# B&R Automation Studio project SortingStation
Automation Studio 4.12.7.113 SP; Project implementing the sorting station of the cap processing machine; technology packages: mapp 5.24.3, mappCockpit 5.24.4, mappMotion 5.24.1, mappView 5.24.4

## Configuration SortingStation

CPU 5PPC2100.BY44-000, AutomationRuntime I4.83, Build 4.1.2, Safety 0.0, Vc V4.73.2

### Task classes (Cpu.sw)
```
Cyclic#1 (cycle 2000 us, tolerance 0 us):
  Conveyor <- Source.Conveyor.Conveyor.prg
Cyclic#4:
  Comms <- Infrastructure.Comms.Comms.prg
  Automatic <- Source.Automatic.Automatic.prg
  ManualMode <- Source.Manual.ManualMode.prg
  Homing <- Source.Homing.Homing.prg
  Sorter <- Source.Sorter.Sorter.prg
Cyclic#8:
  Recipe <- Infrastructure.Recipe.Recipe.prg
  AlarmHandl <- Infrastructure.Alarms.AlarmHandling.prg
  HMIHelper <- Infrastructure.HMIHelper.HMIHelper.prg
DataObjects: McAcpSys
NcDataObjects: McDriveLog
Binaries: McAcpDrv, udbdef, McAcpSim, mvLoader, arflatprv, McProfGen, mCoWebSc, TCData, FWRules, arcoal, arsvcreg, iomap, asfw, Role, ashwac, sysconf, arconfig, SortConv, ashwd, User, SortRecipe, SortAlaCor, SortSett, SortAlaHis, Settings, Config
Libraries: CoTrace, AsZip, FileIO, runtime, McBase, MpBase, AsOpcUac, AsOpcUas, McAcpAx, McAxis, McStpAx, MpAxis, MpRecipe, sys_lib, MpFile, standard, MpAlarmX, astime, MpServer, asieccon, asbrstr, asio, asepl, asioacc, asusb, arssl, powerlnk, dataobj, aruser
```

### Hardware
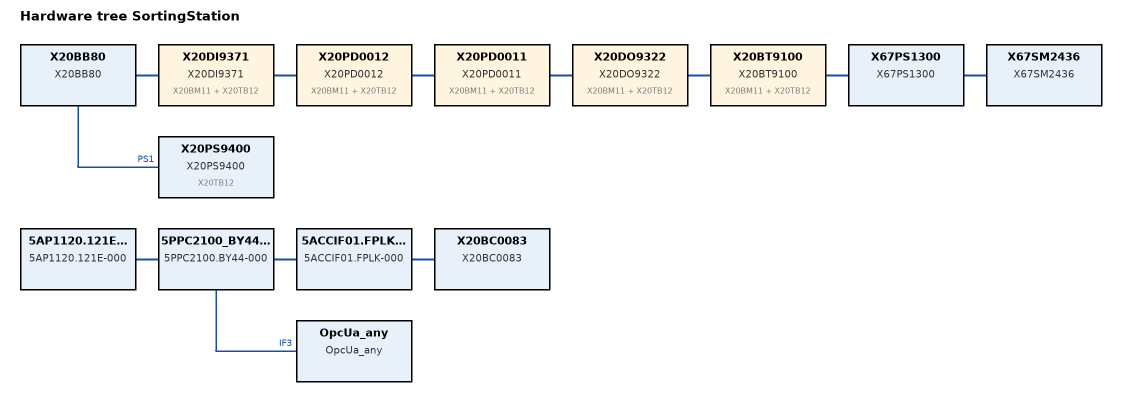
```
5ACCIF01.FPLK-000 : 5ACCIF01.FPLK-000 v1.7.1.0  [SL -> 5PPC2100_BY44_000.SL1]
  Connector IF1:
    ActivateANSL = 1
5AP1120.121E-000 : 5AP1120.121E-000 v2.0.0.0
5PPC2100_BY44_000 : 5PPC2100.BY44-000 v2.1.1.0  [SY -> 5AP1120.121E-000.SY1]
  Connector IF3:
    AssignedOperatingSystem = ARemb
    ActivateDevice = 1
    HostName = sorting-station-ppc2100
    ActivateSnmp = 2
  Connector IF4:
    AssignedOperatingSystem = GPOS
  Connector IF7:
    OperatingSystem = ARemb
    ActivateDevice = 1
    HostName = sorting-station-ppc2100
    Mode = Manual
    InternetAddress = 192.169.0.10
    SubnetMask = 255.255.255.0
    ActivateSnmp = 2
  Connector IF5:
    AssignedOperatingSystem = ARemb
  Connector IF6:
    AssignedOperatingSystem = GPOS
  ConfigurationID = SortingStation_SortingStation
  Cyclic1Duration = 2000
  Cyclic1Tolerance = 0
  FileDevice1
  FileDeviceName1 = USER
  FileDevicePath1 = C:/recipe
  TimeZone = 65
  ActivateDaylightSavingTime = 1
  FtpUser1
  FtpUsername1 = admin  // admin
  FtpUserPassword1 = UdIKPno0znT3css1/ZU0JOxNTb+d8jjj3jhTbXr/0FY=  // admin
  FtpUserSalt1 = m5VJdN1Q
  FTPAccessRight1 = 0
  FTPdevice1 = ALL
  ActivateOpcUa = 1
  OpcUaInformationModels_PV_Version = 1
  ActivateHypervisor = 1
  ARembDramSizeInMb = 512
OpcUa_any : OpcUa_any v1.0.0.1  [ETH1 -> 5PPC2100_BY44_000.IF3 [Cable Type=PowerlinkCable, Length=10, Version=1.0.0.3]]
  ServerDiagnostics = on
  ServerEndpointUrl = opc.tcp://10.67.22.6:4840
  Channel1
  ChannelID1 = ProductAtUnloadingPosition  // Bit from Distribution Station signaling the product is arriving
  ChannelBrowsePath1 = /0:Root/0:Objects/4:PLC/6:Modules/6:&:&:/6:Global PV/6:IO/6:DIn/6:ProductAtUnloadingPosition  // Browse path for the OPCUA node
  Channel2
  ChannelID2 = DistributionReady  // Variable received from Distribution signaling it is ready (no errors)
  ChannelBrowsePath2 = /0:Root/0:Objects/4:PLC/6:Modules/6:&:&:/6:Global PV/6:MachineControl/6:Status/6:ReadyToRun  // Browse path for the OPCUA node
X20BB80 : X20BB80 v1.1.0.0
X20BC0083 : X20BC0083 v2.14.0.0  [PLK1 -> 5ACCIF01.FPLK-000.IF1 (NodeNumber=1) [Cable Type=PowerlinkCable, Length=10, Version=1.0.0.3]; SL -> X20BB80.SL1]
  Supervision = off
X20BM11 : X20BM11 v1.1.0.0  [X2X1 -> X20BB80.IF1]
X20BM11a : X20BM11 v1.1.0.0  [X2X1 -> X20BM11.X2X2]
X20BM11b : X20BM11 v1.1.0.0  [X2X1 -> X20BM11a.X2X2]
X20BM11c : X20BM11 v1.1.0.0  [X2X1 -> X20BM11b.X2X2]
X20BM11d : X20BM11 v1.1.0.0  [X2X1 -> X20BM11c.X2X2]
X20BT9100 : X20BT9100 v1.3.0.0  [SS1 -> X20TB12e.SS; SL -> X20BM11d.SL1]
  Supervision = off
X20DI9371 : X20DI9371 v1.4.0.0  [SS1 -> X20TB12a.SS; SL -> X20BM11.SL1]
  Supervision = off
X20DO9322 : X20DO9322 v1.5.0.0  [SS1 -> X20TB12d.SS; SL -> X20BM11c.SL1]
  Supervision = off
X20PD0011 : X20PD0011 v1.2.0.0  [SS1 -> X20TB12c.SS; SL -> X20BM11b.SL1]
  Supervision = off
X20PD0012 : X20PD0012 v1.2.0.0  [SS1 -> X20TB12b.SS; SL -> X20BM11a.SL1]
  Supervision = off
X20PS9400 : X20PS9400 v1.8.0.0  [SS1 -> X20TB12.SS; PS -> X20BB80.PS1]
  Supervision = off
X20TB12 : X20TB12 v1.0.0.0
X20TB12a : X20TB12 v1.0.0.0
X20TB12b : X20TB12 v1.0.0.0
X20TB12c : X20TB12 v1.0.0.0
X20TB12d : X20TB12 v1.0.0.0
X20TB12e : X20TB12 v1.0.0.0
X67PS1300 : X67PS1300 v1.0.0.0  [X2X1 -> X20BT9100.X2X1 [Cable Type=X2XCable, Length=10, Version=1.0.0.3]]
X67SM2436 : X67SM2436 v2.3.0.0  [X2X1 -> X67PS1300.X2X2 [Cable Type=X2XCable, Length=10, Version=1.0.0.3]]
  Supervision = off
  FunctionModel/DriveConfiguration/Module:
    ActivateModuleSimulationOnPLC = Off
  FunctionModel/DriveConfiguration:
    ModuleParameters = StepperParameters
  FunctionModel/DriveConfiguration/ModuleParameters:
    McStepperTypeID = X67Config
    EncoderType = Incremental
    ReferencePulse = yes
    RatedCurrent = 3.0
    MaximumCurrent = 5.01
    AxesNumber = 2
    FullStepThreshold = 1
    StallDetection = 1
    SmartCurrentControl = 0
    BrakeOutput = 0
    NumberOfDigitalInputs = 6
    NumberOfTriggers = 1
  FunctionModel/DriveConfiguration/Channel[1]/RealAxis:
    AxisReference = gAxisSort
  FunctionModel/DriveConfiguration/Channel[1]/RealAxis/MechanicalElements/Gearbox:
    InputIsReadOnly = 0
    Input = 1
    OutputIsReadOnly = 0
    Output = 1
  FunctionModel/DriveConfiguration/Channel[1]/RealAxis/MechanicalElements/RotaryToLinearTransformation:
    ReferenceDistanceIsReadOnly = 0
    ReferenceDistance = 4
  FunctionModel/DriveConfiguration/Channel[1]/RealAxis/Motor:
    SteppingAngle = 1.8
  FunctionModel/DriveConfiguration/Channel[1]/RealAxis:
    EncoderLink = NoEncoder
  FunctionModel/DriveConfiguration/Channel[1]/RealAxis/Controller:
    ModeIsReadOnly = 0
    Mode = CurrentController
  FunctionModel/DriveConfiguration/Channel[1]/RealAxis/Controller/Mode/Current:
    StandstillCurrent = 1.5
    ConstantSpeedCurrent = 1.5
    SpeedChangeCurrent = 1.5
    FullStepThreshold = 0
    MotorSettlingTime = 1
    DelayedCurrentSwitchOff = 1
  FunctionModel/DriveConfiguration/Channel[1]/RealAxis/Homing:
    Mode = Direct
  FunctionModel/DriveConfiguration/Channel[1]/RealAxis/Homing/Mode:
    Position = 0.0
    ReferencePulse = NotUsed
  FunctionModel/DriveConfiguration/Channel[1]/RealAxis/Homing:
    RestorePositionVariable = 
    ClearPositionError = No
  FunctionModel/DriveConfiguration/Channel[1]/RealAxis/StopReaction:
    DriveError = DecelerationLimit
  FunctionModel/DriveConfiguration/Channel[1]/RealAxis/MovementErrorLimits:
    PositionError = 1.0
    StallDetectionConfiguration = NotUsed
  FunctionModel/DriveConfiguration/Channel[1]/RealAxis:
    JerkFilter = NotUsed
    ZeroVibrationFilter = NotUsed
  FunctionModel/DriveConfiguration/Channel[1]/RealAxis/DigitalInputs/HomingSwitch:
    Source = NotUsed
    Level = High
  FunctionModel/DriveConfiguration/Channel[1]/RealAxis/DigitalInputs/PositiveLimitSwitch:
    Source = NotUsed
    Level = High
  FunctionModel/DriveConfiguration/Channel[1]/RealAxis/DigitalInputs/NegativeLimitSwitch:
    Source = NotUsed
    Level = High
  FunctionModel/DriveConfiguration/Channel[1]/RealAxis/DigitalInputs/Trigger1:
    Source = NotUsed
    Level = High
  FunctionModel/DriveConfiguration/Channel[1]/RealAxis/DigitalInputs/Trigger2:
    Source = NotUsed
    Level = High
  FunctionModel/DriveConfiguration/Channel[1]/RealAxis/DigitalInputs/Quickstop:
    Input = NotUsed
  FunctionModel/DriveConfiguration/Channel[1]/RealAxis/DigitalOutputs:
    BrakeControl = NotUsed
  FunctionModel/DriveConfiguration/Channel[1]/RealAxis/Simulation:
    LoadSimulationMode = NotUsed
  FunctionModel/DriveConfiguration/Channel[2]/RealAxis:
    AxisReference = 
  FunctionModel/DriveConfiguration/Channel[2]/RealAxis/MechanicalElements/Gearbox:
    InputIsReadOnly = 0
    Input = 1
    OutputIsReadOnly = 0
    Output = 1
  FunctionModel/DriveConfiguration/Channel[2]/RealAxis/MechanicalElements/RotaryToLinearTransformation:
    ReferenceDistanceIsReadOnly = 0
    ReferenceDistance = 1
  FunctionModel/DriveConfiguration/Channel[2]/RealAxis/Motor:
    SteppingAngle = 1.8
  FunctionModel/DriveConfiguration/Channel[2]/RealAxis:
    EncoderLink = NoEncoder
  FunctionModel/DriveConfiguration/Channel[2]/RealAxis/Controller:
    ModeIsReadOnly = 0
    Mode = CurrentController
  FunctionModel/DriveConfiguration/Channel[2]/RealAxis/Controller/Mode/Current:
    StandstillCurrent = 0.09
    ConstantSpeedCurrent = 0.45
    SpeedChangeCurrent = 0.9
    FullStepThreshold = 0.0
    MotorSettlingTime = 1
    DelayedCurrentSwitchOff = 1
  FunctionModel/DriveConfiguration/Channel[2]/RealAxis/Homing:
    Mode = Direct
  FunctionModel/DriveConfiguration/Channel[2]/RealAxis/Homing/Mode:
    Position = 0.0
    ReferencePulse = NotUsed
  FunctionModel/DriveConfiguration/Channel[2]/RealAxis/Homing:
    RestorePositionVariable = 
    ClearPositionError = No
  FunctionModel/DriveConfiguration/Channel[2]/RealAxis/StopReaction:
    DriveError = DecelerationLimit
  FunctionModel/DriveConfiguration/Channel[2]/RealAxis/MovementErrorLimits:
    PositionError = 1.0
    StallDetectionConfiguration = NotUsed
  FunctionModel/DriveConfiguration/Channel[2]/RealAxis:
    JerkFilter = NotUsed
    ZeroVibrationFilter = NotUsed
  FunctionModel/DriveConfiguration/Channel[2]/RealAxis/DigitalInputs/HomingSwitch:
    Source = NotUsed
    Level = High
  FunctionModel/DriveConfiguration/Channel[2]/RealAxis/DigitalInputs/PositiveLimitSwitch:
    Source = NotUsed
    Level = High
  FunctionModel/DriveConfiguration/Channel[2]/RealAxis/DigitalInputs/NegativeLimitSwitch:
    Source = NotUsed
    Level = High
  FunctionModel/DriveConfiguration/Channel[2]/RealAxis/DigitalInputs/Trigger1:
    Source = NotUsed
    Level = High
  FunctionModel/DriveConfiguration/Channel[2]/RealAxis/DigitalInputs/Trigger2:
    Source = NotUsed
    Level = High
  FunctionModel/DriveConfiguration/Channel[2]/RealAxis/DigitalInputs/Quickstop:
    Input = NotUsed
  FunctionModel/DriveConfiguration/Channel[2]/RealAxis/DigitalOutputs:
    BrakeControl = NotUsed
  FunctionModel/DriveConfiguration/Channel[2]/RealAxis/Simulation:
    LoadSimulationMode = NotUsed
```

### IoMap.iom - 5PPC2100_BY44_000/IoMap.iom
```iecst
VAR_CONFIG
	::gSorterHardwareIO.DigitalInputs.diProdAvail AT %IX."X20DI9371".DigitalInput01; (*24 VDC, 0.1 to 25 ms switching delay, sink - Product available*)
	::gSorterHardwareIO.DigitalInputs.diMetallic AT %IX."X20DI9371".DigitalInput02; (*24 VDC, 0.1 to 25 ms switching delay, sink - Product is metallic*)
	::gSorterHardwareIO.DigitalInputs.diNotBlack AT %IX."X20DI9371".DigitalInput03; (*24 VDC, 0.1 to 25 ms switching delay, sink - Product is not black*)
	::gSorterHardwareIO.DigitalInputs.diLaneFull AT %IX."X20DI9371".DigitalInput04; (*24 VDC, 0.1 to 25 ms switching delay, sink - Lane full*)
	::gSorterHardwareIO.DigitalInputs.diSwitch1Retracted AT %IX."X20DI9371".DigitalInput05; (*24 VDC, 0.1 to 25 ms switching delay, sink - Switch 1 retracted*)
	::gSorterHardwareIO.DigitalInputs.diSwitch1Extended AT %IX."X20DI9371".DigitalInput06; (*24 VDC, 0.1 to 25 ms switching delay, sink - Switch 1 extended*)
	::gSorterHardwareIO.DigitalInputs.diSwitch2Retracted AT %IX."X20DI9371".DigitalInput07; (*24 VDC, 0.1 to 25 ms switching delay, sink - Switch 2 retracted*)
	::gSorterHardwareIO.DigitalInputs.diSwitch2Extended AT %IX."X20DI9371".DigitalInput08; (*24 VDC, 0.1 to 25 ms switching delay, sink - Switch 2 extended*)
	::gSorterHardwareIO.DigitalOutputs.doExtendSwitch1 AT %QX."X20DO9322".DigitalOutput02; (*24 VDC / 0.5 A, source - Extend switch 1*)
	::gSorterHardwareIO.DigitalOutputs.doExtendSwitch2 AT %QX."X20DO9322".DigitalOutput03; (*24 VDC / 0.5 A, source - Extend switch 2*)
	::gSorterHardwareIO.DigitalOutputs.doRetractStopper AT %QX."X20DO9322".DigitalOutput04; (*24 VDC / 0.5 A, source - Retract stopper*)
	::AlarmHandl:CommsErrors.PLK.FPLK_ModuleOk AT %IX."5ACCIF01.FPLK-000".ModuleOk;
	::AlarmHandl:CommsErrors.X2X.X20BC0083_ModuleOk AT %IX."X20BC0083".ModuleOk;
	::AlarmHandl:CommsErrors.X2X.X20PS9400_ModuleOk AT %IX."X20PS9400".ModuleOk;
	::AlarmHandl:CommsErrors.X2X.X20DI9371_ModuleOk AT %IX."X20DI9371".ModuleOk;
	::AlarmHandl:CommsErrors.X2X.X20PD0012_ModuleOk AT %IX."X20PD0012".ModuleOk;
	::AlarmHandl:CommsErrors.X2X.X20PD0011_ModuleOk AT %IX."X20PD0011".ModuleOk;
	::AlarmHandl:CommsErrors.X2X.X20DO9322_ModuleOk AT %IX."X20DO9322".ModuleOk;
	::AlarmHandl:CommsErrors.X2X.X20BT9100_ModuleOk AT %IX."X20BT9100".ModuleOk;
	::AlarmHandl:CommsErrors.X2X.X67SM2436_ModuleOk AT %IX."X67SM2436".ModuleOk;
	::OpcUaControl.Read.ProductArriving AT %IX."OpcUa_any".ProductAtUnloadingPosition; (*Signal that product is arriving from the distribution station*)
	::OpcUaControl.Read.DistributionReady AT %IX."OpcUa_any".DistributionReady; (*Signal that distribution is without errors and ready to go*)
END_VAR
```

- Physical/SortingStation/5PPC2100_BY44_000/PvMap.vvm: same as Physical/SortingStation/5PPC2100_BY44_000/Cpu.per
### SortConv.axis - 5PPC2100_BY44_000/mappMotion/SortConv.axis
```
Element gAxisSort (Type=axis)
  BaseTypeIsReadOnly = 0
  BaseType = Rotary
    MeasurementUnitIsReadOnly = 0
    MeasurementUnit = 17476
    MeasurementResolutionIsReadOnly = 0
    MeasurementResolution = 0.01
    CountDirectionIsReadOnly = 0
    CountDirection = Standard
  MovementLimitsIsReadOnly = 0
  MovementLimits = Internal
    Position:
      LowerLimitMin = -1.79769313486231E308
      UpperLimitMax = 1.79769313486231E308
      LowerLimit = -1000.0
      UpperLimit = 1000.0
    VelocityIsReadOnly = 0
    Velocity:
      VelocityMax = 3.4E38
      Velocity = 1000
    AccelerationIsReadOnly = 0
    Acceleration:
      AccelerationMax = 3.4E38
      Acceleration = 5000
    DecelerationIsReadOnly = 0
    Deceleration:
      DecelerationMax = 3.4E38
      Deceleration = 5000
  Alarms = None
```

### SortAlaCor.mpalarmxcore - 5PPC2100_BY44_000/mappServices/Alarm/SortAlaCor.mpalarmxcore
```
Element MpLinkSORTING_gAlarmXCore (Type=mpalarmxcore)
  mapp.AlarmX.Core.Configuration:
    [0]:
      Name = Sorting station not homed
      Message = Cannot start automtic mode, the machine needs to be homed first.
      Code = 1001
      Behavior = DiscreteValueMonitoring
        Monitoring:
          MonitoredPV = ::AlarmHandl:CommsErrors.X2X.X20BC0083_ModuleOk
          TriggerValues:
            [0] = FALSE
    [1]:
      Name = Automatic in Error state
      Message = The automatic flow has been stopped, error is present. Please clear error and then re-home machine.
      Code = 1002
    [2]:
      Name = Product stuck between stopper and lane
      Message = The product did not reach the lane, please remove the product and re-home the machine.
      Code = 2001
      Behavior = PersistentAlarm
    [3]:
      Name = Product behind stopper
      Message = Either a second product has come up, or the product did not make it through the stopper after being identified. Please remove the product and rehome the machine.
      Code = 2002
    [4]:
      Name = Incorrect switch open
      Message = If a product is present, you cannot open the correct stopper until the right switch is open. Please see guidelines and try again.
      Code = 3001
    [5]:
      Name = PLK comms error
      Message = There was an error communicating over Powerlink. Please check PLK card and cable connection.
      Code = 4001
    [6]:
      Name = X2X comms error
      Message = There was an error communicating with one of the X20 or X67 modules. Please check connections.
      Code = 4002
    [7]:
      Name = OPCUA comms error
      Message = There was an error in the OPCUA connection. Please check the parameters and re-attempt connection.
```

### SortAlaHis.mpalarmxhistory - 5PPC2100_BY44_000/mappServices/Alarm/SortAlaHis.mpalarmxhistory
```
Element MpLinkSORTING_gAlarmXHistory (Type=mpalarmxhistory)
```

### SortRecipe.mprecipexml - 5PPC2100_BY44_000/mappServices/Recipe/SortRecipe.mprecipexml
```
Element MpLinkSORTING_gRecipeXml (Type=mprecipexml)
```

## Logical view

Binary libraries used (declarations not repeated): operator, runtime, astime, AsIecCon, CoTrace 5.24.4, AsZip, FileIO, McBase 5.24.1, MpBase 5.24.1, AsOpcUac, AsOpcUas, McAcpAx 5.24.1, McAxis 5.24.1, McStpAx 5.24.1, MpAxis 5.24.1, MpRecipe 5.24.3, sys_lib, MpFile 5.24.3, standard, MpAlarmX 5.24.3, MpServer 5.24.0

### Global.typ - Global data types
```iecst
(*global enums*)

TYPE
	gOperatingModeType : 	STRUCT  (*Type for tracking the mode'*)
		AutoMode : BOOL; (*Automatic mode*)
		ManualMode : BOOL; (*Manual mode*)
		HomingMode : BOOL; (*Homing mode*)
	END_STRUCT;
	gOperatingModeEnum :
		( (*Global operating mode*)
		AUTOMATIC := 1, (*Automatic running mode*)
		MANUAL := 2, (*Manual operation mode*)
		HOMING := 3 (*Homing mode*)
		);
END_TYPE

(*global types for sorter hardware*)

TYPE
	gSorterDOType : 	STRUCT  (*Sorter digital output type*)
		doExtendSwitch1 : BOOL; (*Command to extend switch 1*)
		doExtendSwitch2 : BOOL; (*Command to extend switch 2*)
		doRetractStopper : BOOL; (*Retract the stopper*)
	END_STRUCT;
	gSorterDIType : 	STRUCT  (*Sorter digital input type*)
		diProdAvail : BOOL; (*Product available*)
		diMetallic : BOOL; (*Product is metallic*)
		diNotBlack : BOOL; (*Product is not black*)
		diLaneFull : BOOL; (*Lane is full of a product*)
		diSwitch1Retracted : BOOL; (*Switch 1 is retracted*)
		diSwitch1Extended : BOOL; (*Switch 1 is extended*)
		diSwitch2Retracted : BOOL; (*Switch 2 is retracted*)
		diSwitch2Extended : BOOL; (*Switch 2 is extended*)
	END_STRUCT;
	gSorterHardwareIOType : 	STRUCT  (*Hardware IO structure*)
		DigitalOutputs : gSorterDOType; (*Digital outputs*)
		DigitalInputs : gSorterDIType; (*Digital inputs*)
	END_STRUCT;
END_TYPE
```

### Global.var - Global variables
```iecst
(*global variables*)
VAR
	gOperatingMode : gOperatingModeType; (*Mode of operation of the sorting station*)
END_VAR
(*global interface for hardware connect*)
VAR
	gSorterHardwareIO : gSorterHardwareIOType; (*Hardware object for the sorter*)
END_VAR
(*control buttons from main page*)
VAR
	gReset : BOOL; (*Reset/clear button*)
	gStop : BOOL; (*Stop button*)
	gStart : BOOL; (*Start button for the chosen operating mode*)
END_VAR
```


### Package Logical/Source - Package for source code

### Package Logical/Source/Manual - Package for manual mode source code

### ManualIF.typ - Manual interface types
```iecst
(*global interface types*)

TYPE
	ManualCommandType : 	STRUCT  (*Commands type for manual mode*)
		ClassifyProduct : BOOL; (*Command to classify product*)
		JogConveyorBackward : BOOL; (*Jog conveyor forward*)
		JogConveyorForward : BOOL; (*Jog conveyor backward*)
		RetractStopper : BOOL; (*Retract stopper*)
		ExtendSwitch2 : BOOL; (*Extend switch 1*)
		ExtendSwitch1 : BOOL; (*Extend switch 2*)
	END_STRUCT;
	ManualControlType : 	STRUCT  (*Manual mode control structure type*)
		Cmd : ManualCommandType; (*Command for manual mode*)
		Status : ManualStatusType; (*Status for manual mode*)
	END_STRUCT;
	ManualStatusType : 	STRUCT  (*Status type for manual mode*)
		ProductClassified : BOOL; (*Status showing product has been classified*)
		DestinationLane : USINT; (*Lane 1, 2 or 3 - default is 3*)
		ProductInActiveArea : BOOL; (*True if the product is between stopper and lane*)
		Error : BOOL; (*Error triggered*)
	END_STRUCT;
END_TYPE
```

### ManualIF.var - Manual interface variables
```iecst
(*global interface variables*)
VAR
	ManualControl : ManualControlType; (*Control structure for manual mode*)
END_VAR
```

### Program Logical/Source/Manual/ManualMode (IEC) - Manual mode program

#### Cyclic.ld - Cyclic code
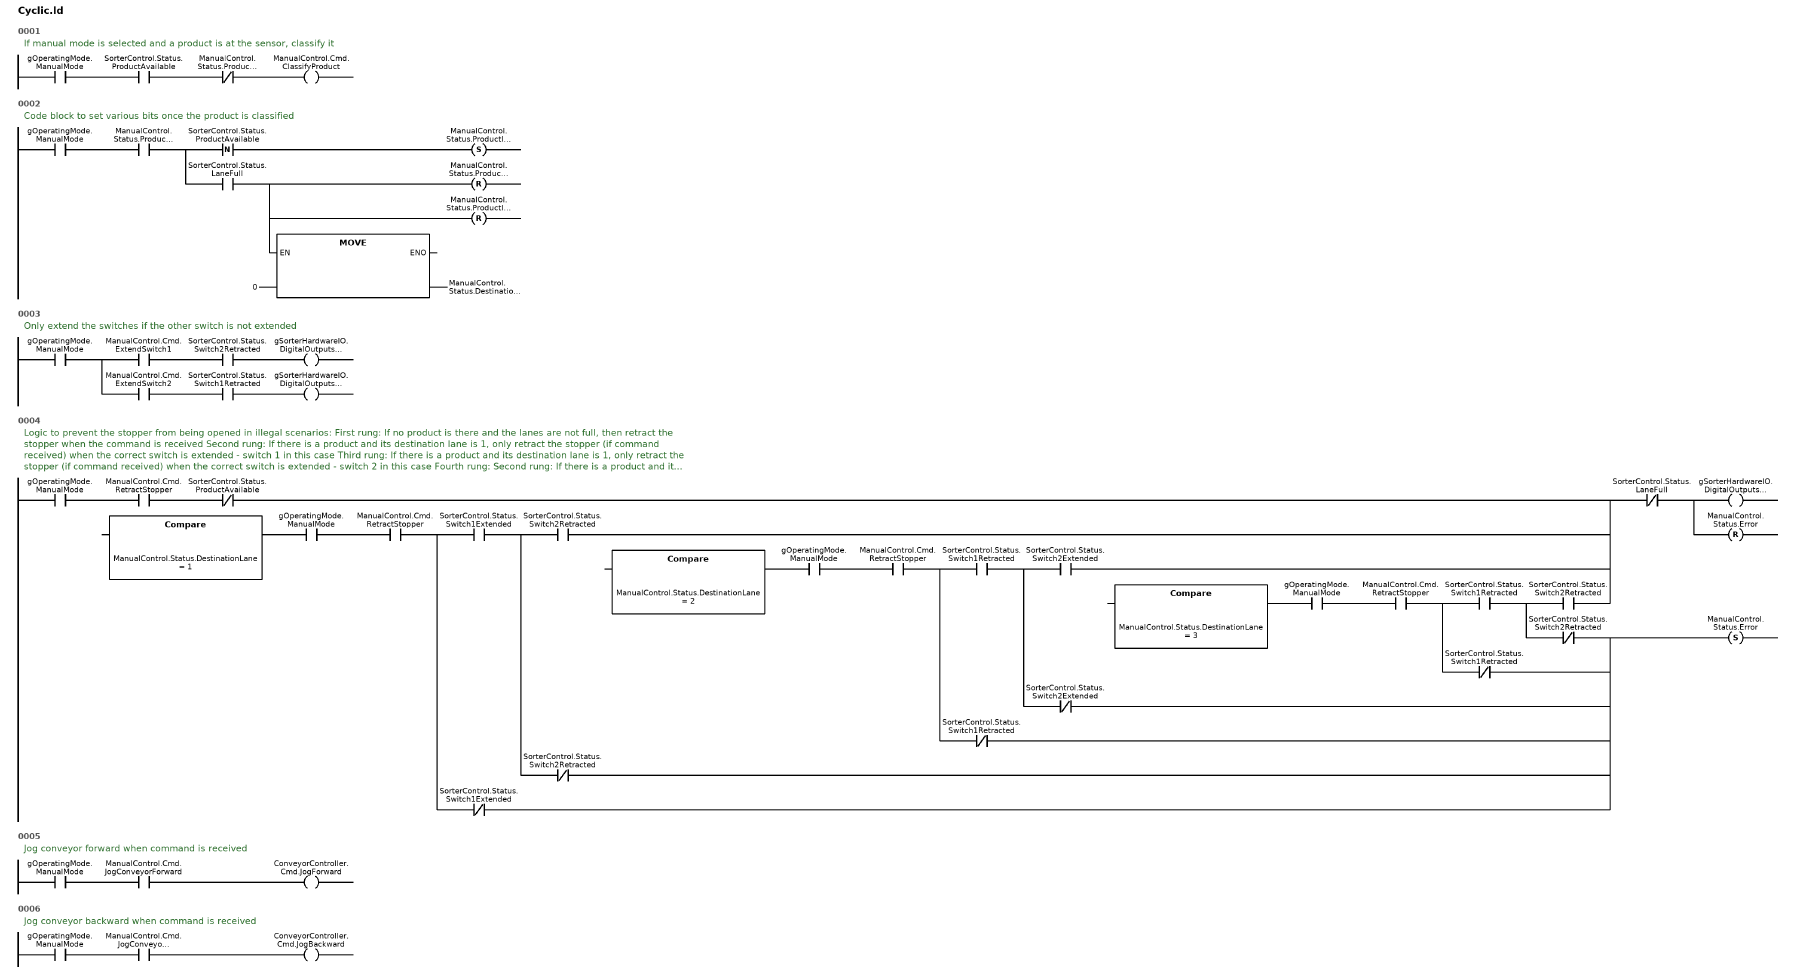
Ladder, written as Structured Text:
```iecst
PROGRAM _CYCLIC
VAR
    _p1 : BOOL;
    _e2 : F_TRIG;
    _p3 : BOOL;
    _p4 : BOOL;
    _p5 : BOOL;
    _p6 : BOOL;
END_VAR
(* Network 1: If manual mode is selected and a product is at the sensor, classify it *)
ManualControl.Cmd.ClassifyProduct := gOperatingMode.ManualMode AND SorterControl.Status.ProductAvailable AND NOT ManualControl.Status.ProductClassified;

(* Network 2: Code block to set various bits once the product is classified *)
_p1 := gOperatingMode.ManualMode AND ManualControl.Status.ProductClassified;
_e2(CLK := SorterControl.Status.ProductAvailable);
IF _p1 AND _e2.Q THEN ManualControl.Status.ProductInActiveArea := TRUE; END_IF;
IF _p1 AND SorterControl.Status.LaneFull THEN
    ManualControl.Status.ProductClassified := FALSE;
    ManualControl.Status.ProductInActiveArea := FALSE;
    ManualControl.Status.DestinationLane := 0;
END_IF;

(* Network 3: Only extend the switches if the other switch is not extended *)
gSorterHardwareIO.DigitalOutputs.doExtendSwitch1 := gOperatingMode.ManualMode AND ManualControl.Cmd.ExtendSwitch1 AND SorterControl.Status.Switch2Retracted;
gSorterHardwareIO.DigitalOutputs.doExtendSwitch2 := gOperatingMode.ManualMode AND ManualControl.Cmd.ExtendSwitch2 AND SorterControl.Status.Switch1Retracted;

(* Network 4: Logic to prevent the stopper from being opened in illegal scenarios: First rung: If no product is there and the lanes are not full, then retract the stopper when the command is received Second rung: If there is a product and its destination lane is 1, only retract the stopper (if command received) when the correct switch is extended - switch 1 in this case Third rung: If there is a product and its destination lane is 1, only retract the stopper (if command received) when the correct switch is extended - switch 2 in this case Fourth rung: Second rung: If there is a product and its destination lane is 1, only retract the stopper (if command received) when no switches are extended Trigger an error in other cases *)
_p3 := (ManualControl.Status.DestinationLane = 1) AND gOperatingMode.ManualMode AND ManualControl.Cmd.RetractStopper;
_p4 := (ManualControl.Status.DestinationLane = 2) AND gOperatingMode.ManualMode AND ManualControl.Cmd.RetractStopper;
_p5 := (ManualControl.Status.DestinationLane = 3) AND gOperatingMode.ManualMode AND ManualControl.Cmd.RetractStopper;
_p6 := ((gOperatingMode.ManualMode AND ManualControl.Cmd.RetractStopper AND NOT SorterControl.Status.ProductAvailable) OR (_p3 AND SorterControl.Status.Switch1Extended AND SorterControl.Status.Switch2Retracted) OR (_p4 AND SorterControl.Status.Switch1Retracted AND SorterControl.Status.Switch2Extended) OR (_p5 AND SorterControl.Status.Switch1Retracted AND SorterControl.Status.Switch2Retracted)) AND NOT SorterControl.Status.LaneFull;
gSorterHardwareIO.DigitalOutputs.doRetractStopper := _p6;
IF _p6 THEN ManualControl.Status.Error := FALSE; END_IF;
IF (_p5 AND ((SorterControl.Status.Switch1Retracted AND NOT SorterControl.Status.Switch2Retracted) OR NOT SorterControl.Status.Switch1Retracted)) OR (_p4 AND ((SorterControl.Status.Switch1Retracted AND NOT SorterControl.Status.Switch2Extended) OR NOT SorterControl.Status.Switch1Retracted)) OR (_p3 AND ((SorterControl.Status.Switch1Extended AND NOT SorterControl.Status.Switch2Retracted) OR NOT SorterControl.Status.Switch1Extended)) THEN
    ManualControl.Status.Error := TRUE;
END_IF;

(* Network 5: Jog conveyor forward when command is received *)
ConveyorController.Cmd.JogForward := gOperatingMode.ManualMode AND ManualControl.Cmd.JogConveyorForward;

(* Network 6: Jog conveyor backward when command is received *)
ConveyorController.Cmd.JogBackward := gOperatingMode.ManualMode AND ManualControl.Cmd.JogConveyorBackward;
END_PROGRAM
```

#### Init.ld - Initialization code
Ladder, written as Structured Text:
```iecst
PROGRAM _INIT
END_PROGRAM
```

#### Exit.ld - Exit code
Ladder, written as Structured Text:
```iecst
PROGRAM _EXIT
END_PROGRAM
```

### Package Logical/Source/Automatic - Package for automatic source code

### AutomaticIF.typ - Automatic interface types
```iecst
(*global interface types*)

TYPE
	AutomaticCommandType : 	STRUCT  (*Command type for automatic*)
		EnableTimer : BOOL; (*Enable the timer*)
	END_STRUCT;
	AutomaticErrorType : 	STRUCT  (*Errors in automatic mode*)
		Error1 : BOOL; (*ERROR 1 - cannot start automatic mode before homing the station*)
	END_STRUCT;
	AutomaticStatusType : 	STRUCT  (*Status type for automatic*)
		Errors : AutomaticErrorType; (*Errors in Auto mode*)
		SortingReady : BOOL; (*Ready bit for comms*)
	END_STRUCT;
	AutomaticControlType : 	STRUCT  (*Control structure for automatic mode*)
		Cmd : AutomaticCommandType; (*Commands for automatic mode*)
		Status : AutomaticStatusType; (*Status for automatic mode*)
	END_STRUCT;
	AutomaticGeneralInfoType : 	STRUCT  (*General info structure for variables that need to be retained*)
		ProductsTotal : UINT; (*Total number of products*)
		AutomaticModeTime : TIME; (*Time that it has been in automatic mode*)
	END_STRUCT;
END_TYPE
```

### AutomaticIF.var - Automatic interface variables
```iecst
(*global interface variables*)
VAR
	AutomaticController : AutomaticControlType; (*Control structure for Automatic*)
	AutomaticGeneralInfo : AutomaticGeneralInfoType; (*General info that is retained*)
END_VAR
```

### Program Logical/Source/Automatic/Automatic (IEC) - Automatic program

#### Cyclic.ld - Cyclic code
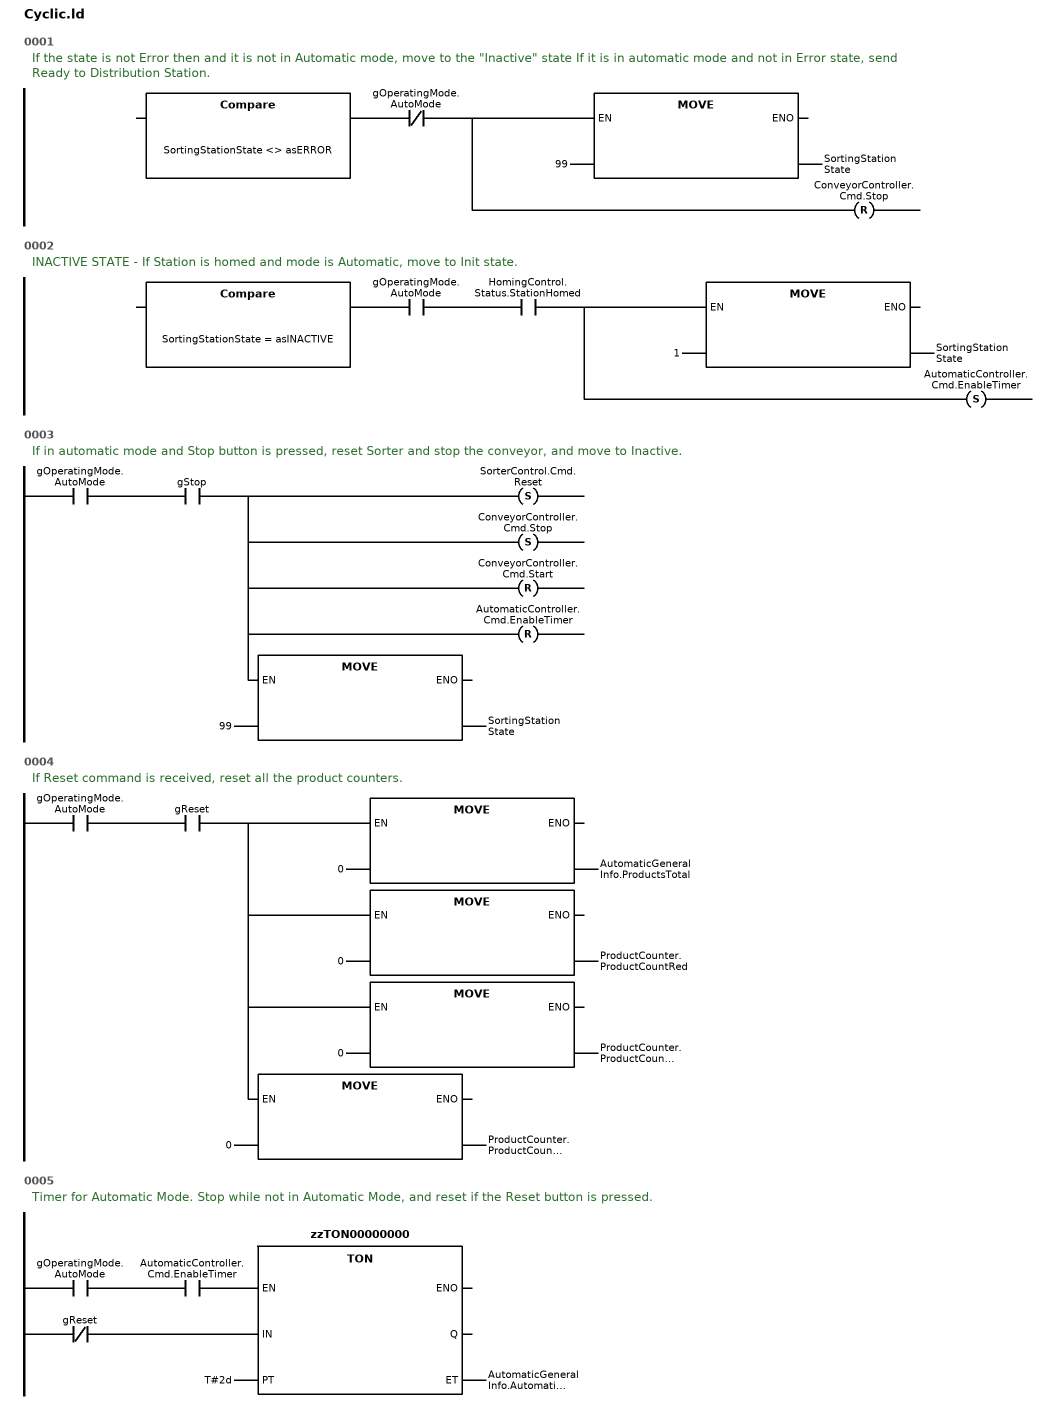
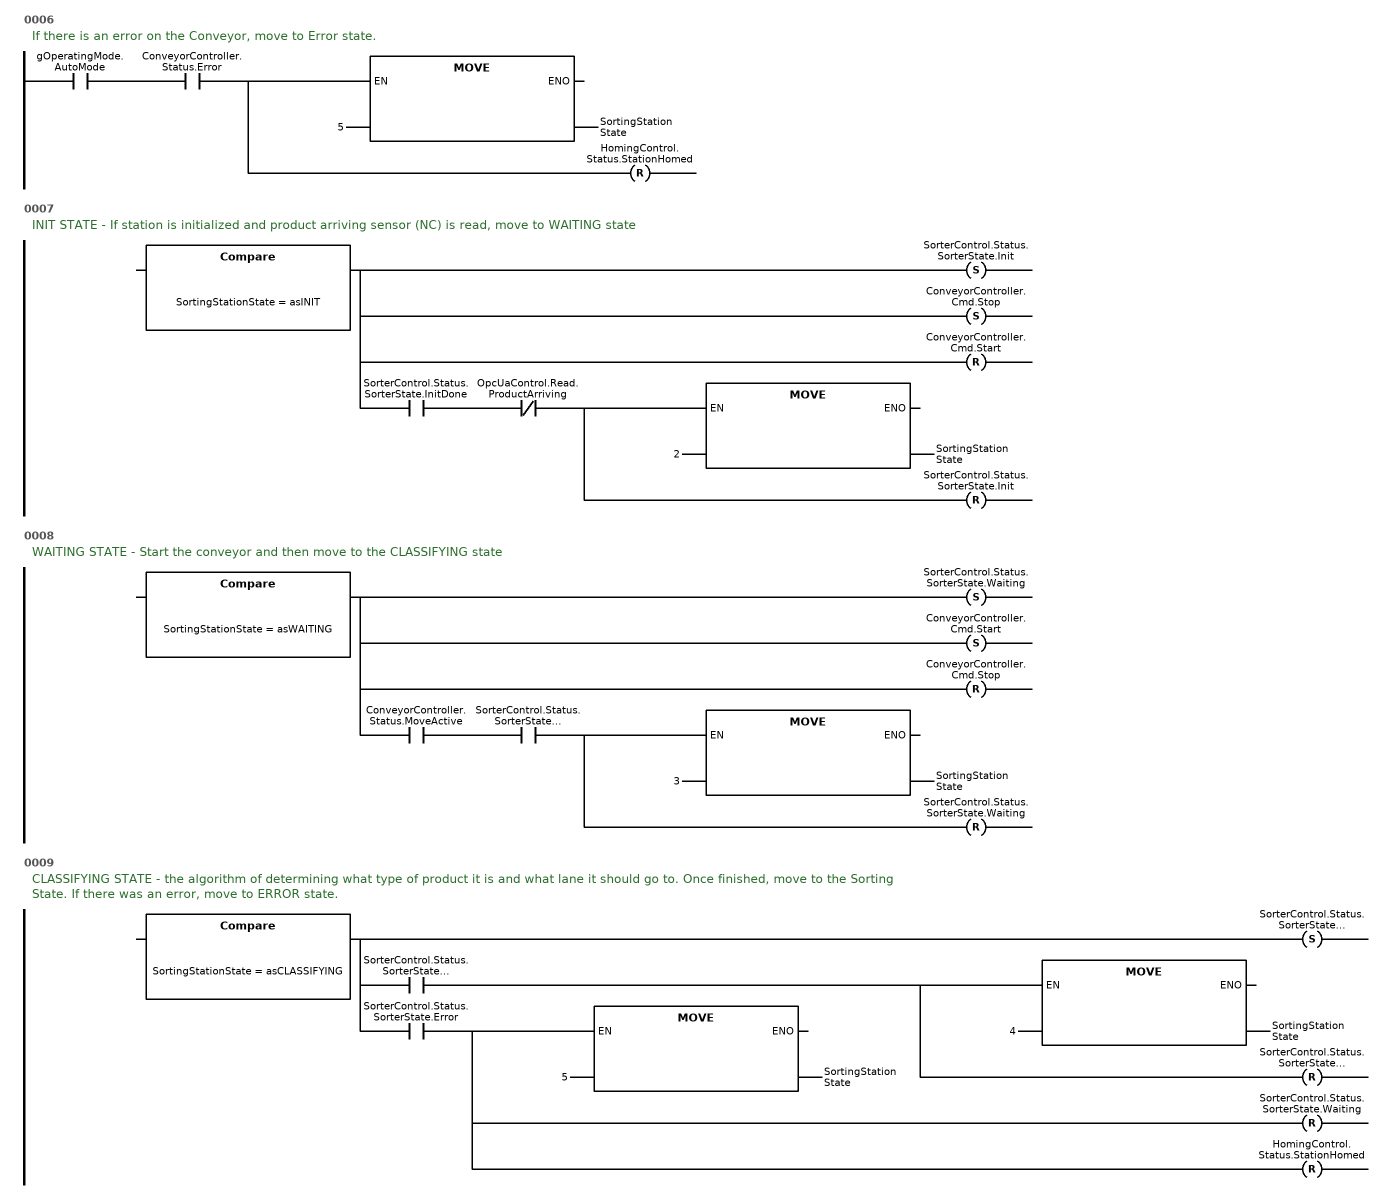
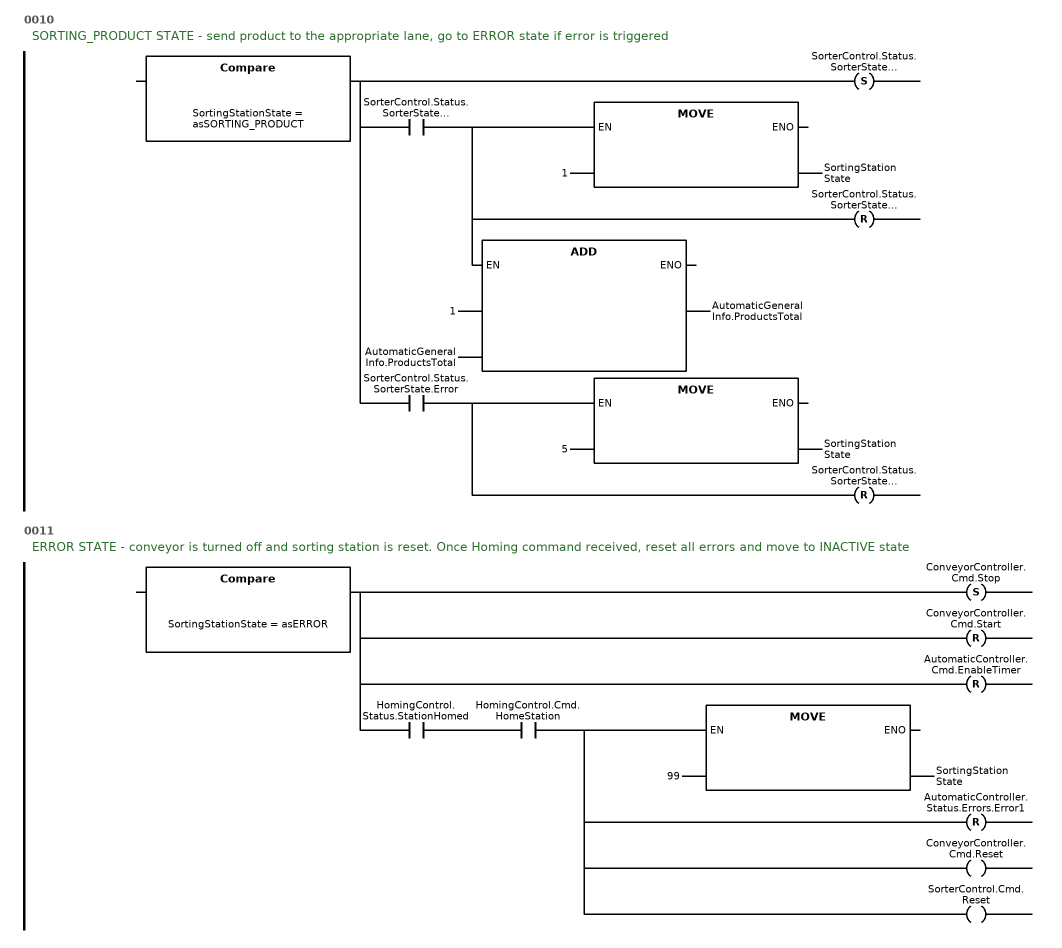
Ladder, written as Structured Text:
```iecst
PROGRAM _CYCLIC
Program to implement state machine for the Automatic Mode
VAR
    _p1 : BOOL;
    _p2 : BOOL;
    _p3 : BOOL;
    _p4 : BOOL;
    _p5 : BOOL;
    _p6 : BOOL;
    _p7 : BOOL;
    _p8 : BOOL;
    _p9 : BOOL;
    _p10 : BOOL;
END_VAR
(* Network 1: If the state is not Error then and it is not in Automatic mode, move to the "Inactive" state If it is in automatic mode and not in Error state, send Ready to Distribution Station. *)
_p1 := (SortingStationState <> asERROR) AND NOT gOperatingMode.AutoMode;
IF _p1 THEN
    SortingStationState := 99;
    ConveyorController.Cmd.Stop := FALSE;
END_IF;

(* Network 2: INACTIVE STATE - If Station is homed and mode is Automatic, move to Init state. *)
_p2 := (SortingStationState = asINACTIVE) AND gOperatingMode.AutoMode AND HomingControl.Status.StationHomed;
IF _p2 THEN
    SortingStationState := 1;
    AutomaticController.Cmd.EnableTimer := TRUE;
END_IF;

(* Network 3: If in automatic mode and Stop button is pressed, reset Sorter and stop the conveyor, and move to Inactive. *)
IF gOperatingMode.AutoMode AND gStop THEN
    SorterControl.Cmd.Reset := TRUE;
    ConveyorController.Cmd.Stop := TRUE;
    ConveyorController.Cmd.Start := FALSE;
    AutomaticController.Cmd.EnableTimer := FALSE;
    SortingStationState := 99;
END_IF;

(* Network 4: If Reset command is received, reset all the product counters. *)
IF gOperatingMode.AutoMode AND gReset THEN
    AutomaticGeneralInfo.ProductsTotal := 0;
    ProductCounter.ProductCountRed := 0;
    ProductCounter.ProductCountBlack := 0;
    ProductCounter.ProductCountMetal := 0;
END_IF;

(* Network 5: Timer for Automatic Mode. Stop while not in Automatic Mode, and reset if the Reset button is pressed. *)
IF gOperatingMode.AutoMode AND AutomaticController.Cmd.EnableTimer THEN
    zzTON00000000(IN := NOT gReset, PT := T#2d);
    AutomaticGeneralInfo.AutomaticModeTime := zzTON00000000.ET;
END_IF;

(* Network 6: If there is an error on the Conveyor, move to Error state. *)
_p3 := gOperatingMode.AutoMode AND ConveyorController.Status.Error;
IF _p3 THEN
    SortingStationState := 5;
    HomingControl.Status.StationHomed := FALSE;
END_IF;

(* Network 7: INIT STATE - If station is initialized and product arriving sensor (NC) is read, move to WAITING state *)
IF (SortingStationState = asINIT) THEN
    SorterControl.Status.SorterState.Init := TRUE;
    ConveyorController.Cmd.Stop := TRUE;
    ConveyorController.Cmd.Start := FALSE;
END_IF;
_p4 := (SortingStationState = asINIT) AND SorterControl.Status.SorterState.InitDone AND NOT OpcUaControl.Read.ProductArriving;
IF _p4 THEN
    SortingStationState := 2;
    SorterControl.Status.SorterState.Init := FALSE;
END_IF;

(* Network 8: WAITING STATE - Start the conveyor and then move to the CLASSIFYING state *)
IF (SortingStationState = asWAITING) THEN
    SorterControl.Status.SorterState.Waiting := TRUE;
    ConveyorController.Cmd.Start := TRUE;
    ConveyorController.Cmd.Stop := FALSE;
END_IF;
_p5 := (SortingStationState = asWAITING) AND ConveyorController.Status.MoveActive AND SorterControl.Status.SorterState.WaitingDone;
IF _p5 THEN
    SortingStationState := 3;
    SorterControl.Status.SorterState.Waiting := FALSE;
END_IF;

(* Network 9: CLASSIFYING STATE - the algorithm of determining what type of product it is and what lane it should go to. Once finished, move to the Sorting State. If there was an error, move to ERROR state. *)
IF (SortingStationState = asCLASSIFYING) THEN
    SorterControl.Status.SorterState.Classifying := TRUE;
END_IF;
_p6 := (SortingStationState = asCLASSIFYING) AND SorterControl.Status.SorterState.ClassifyingDone;
IF _p6 THEN SortingStationState := 4; END_IF;
_p7 := (SortingStationState = asCLASSIFYING) AND SorterControl.Status.SorterState.Error;
IF _p7 THEN SortingStationState := 5; END_IF;
IF _p6 THEN SorterControl.Status.SorterState.Classifying := FALSE; END_IF;
IF _p7 THEN
    SorterControl.Status.SorterState.Waiting := FALSE;
    HomingControl.Status.StationHomed := FALSE;
END_IF;

(* Network 10: SORTING_PRODUCT STATE - send product to the appropriate lane, go to ERROR state if error is triggered *)
IF (SortingStationState = asSORTING_PRODUCT) THEN
    SorterControl.Status.SorterState.SortingProduct := TRUE;
END_IF;
_p8 := (SortingStationState = asSORTING_PRODUCT) AND SorterControl.Status.SorterState.SortingProductDone;
IF _p8 THEN
    SortingStationState := 1;
    SorterControl.Status.SorterState.SortingProduct := FALSE;
    AutomaticGeneralInfo.ProductsTotal := 1 + AutomaticGeneralInfo.ProductsTotal;
END_IF;
_p9 := (SortingStationState = asSORTING_PRODUCT) AND SorterControl.Status.SorterState.Error;
IF _p9 THEN
    SortingStationState := 5;
    SorterControl.Status.SorterState.SortingProduct := FALSE;
END_IF;

(* Network 11: ERROR STATE - conveyor is turned off and sorting station is reset. Once Homing command received, reset all errors and move to INACTIVE state *)
IF (SortingStationState = asERROR) THEN
    ConveyorController.Cmd.Stop := TRUE;
    ConveyorController.Cmd.Start := FALSE;
    AutomaticController.Cmd.EnableTimer := FALSE;
END_IF;
_p10 := (SortingStationState = asERROR) AND HomingControl.Status.StationHomed AND HomingControl.Cmd.HomeStation;
IF _p10 THEN
    SortingStationState := 99;
    AutomaticController.Status.Errors.Error1 := FALSE;
END_IF;
ConveyorController.Cmd.Reset := _p10;
SorterControl.Cmd.Reset := _p10;
END_PROGRAM
```

#### Init.ld - Initialization code
Ladder, written as Structured Text:
```iecst
PROGRAM _INIT
END_PROGRAM
```

#### Exit.ld - Exit code
Ladder, written as Structured Text:
```iecst
PROGRAM _EXIT
END_PROGRAM
```

#### Types.typ - Local data types
```iecst
(*state machine enumerator*)

TYPE
	AutomaticSortingEnum :
		( (*Enum for state machine*)
		asINIT := 1, (*Initial state, homing and setting variables and waiting for start signal*)
		asWAITING := 2, (*Waiting for product to arrive*)
		asCLASSIFYING := 3, (*Identifying and classifying product*)
		asSORTING_PRODUCT := 4, (*Sorting product*)
		asERROR := 5, (*Error state*)
		asINACTIVE := 99
		);
END_TYPE
```

#### Variables.var - Local variables
```iecst
(*local enum*)
VAR
	SortingStationState : AutomaticSortingEnum := asINACTIVE; (*Enumerator to track the state*)
END_VAR
```

### Package Logical/Source/Homing - Package for homing mode

### HomingIF.typ - Homing interface types
```iecst
(*global interface types*)

TYPE
	HomingCommandType : 	STRUCT  (*Commands for homing*)
		HomeStation : BOOL; (*Command to home*)
	END_STRUCT;
	HomingStatusType : 	STRUCT  (*Statuses for homing*)
		StationHomed : BOOL; (*Station is homed*)
	END_STRUCT;
	HomingControlType : 	STRUCT  (*Control structure for homing*)
		Cmd : HomingCommandType; (*Homing commands*)
		Status : HomingStatusType; (*Homing statuses*)
	END_STRUCT;
END_TYPE
```

### HomingIF.var - Homing interface variables
```iecst
(*global interface variables*)
VAR
	HomingControl : HomingControlType; (*Homing controller*)
END_VAR
```

### Program Logical/Source/Homing/Homing (IEC) - Homing task

#### Cyclic.ld - Cyclic code
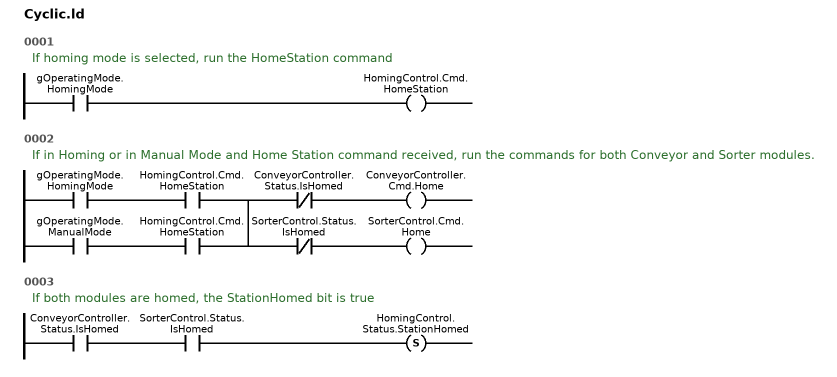
Ladder, written as Structured Text:
```iecst
PROGRAM _CYCLIC
VAR
    _p1 : BOOL;
    _p2 : BOOL;
END_VAR
(* Network 1: If homing mode is selected, run the HomeStation command *)
HomingControl.Cmd.HomeStation := gOperatingMode.HomingMode;

(* Network 2: If in Homing or in Manual Mode and Home Station command received, run the commands for both Conveyor and Sorter modules. *)
_p1 := gOperatingMode.HomingMode AND HomingControl.Cmd.HomeStation;
_p2 := gOperatingMode.ManualMode AND HomingControl.Cmd.HomeStation;
ConveyorController.Cmd.Home := (_p1 OR _p2) AND NOT ConveyorController.Status.IsHomed;
SorterControl.Cmd.Home := (_p1 OR _p2) AND NOT SorterControl.Status.IsHomed;

(* Network 3: If both modules are homed, the StationHomed bit is true *)
IF ConveyorController.Status.IsHomed AND SorterControl.Status.IsHomed THEN
    HomingControl.Status.StationHomed := TRUE;
END_IF;
END_PROGRAM
```

#### Init.ld - Initialization code
Ladder, written as Structured Text:
```iecst
PROGRAM _INIT
END_PROGRAM
```

#### Exit.ld - Exit code
Ladder, written as Structured Text:
```iecst
PROGRAM _EXIT
END_PROGRAM
```

### Package Logical/Source/Conveyor - Package for conveyor source code

### ConveyorIF.typ - Conveyor interface types
```iecst
(*global interface structure types*)

TYPE
	ConveyorCommandType : 	STRUCT  (*Conveyor command structure type*)
		Start : BOOL; (*Command to start the conveyor moving*)
		Stop : BOOL; (*Command to stop the conveyor*)
		Reset : BOOL; (*Command to reset in case of an error*)
		JogForward : BOOL; (*Jog command forward*)
		JogBackward : BOOL; (*Jog command backward*)
		Power : BOOL; (*Command to power on the axis*)
		Home : BOOL; (*Command to home the axis*)
	END_STRUCT;
	ConveyorParameterType : 	STRUCT  (*Conveyor parameter structure type*)
		Position : LREAL := 0.0; (*Initial parameter for the axis - position*)
		Velocity : REAL := 400; (*Initial parameter for the axis - velocity*)
		Acceleration : REAL := 3000; (*Initial parameter for the axis - acceleration*)
		Deceleration : REAL := 3000; (*Initial parameter for the axis - deceleration*)
		HomingMode : McHomingModeEnum := mcHOMING_DEFAULT; (*Homing mode*)
	END_STRUCT;
	ConveyorType : 	STRUCT  (*Conveyor controller type*)
		Cmd : ConveyorCommandType; (*Instance of command structure*)
		Par : ConveyorParameterType; (*Instance of parameter structure*)
		Status : ConveyorStatusType; (*Instance of status structure*)
	END_STRUCT;
	ConveyorStatusType : 	STRUCT  (*Conveyor status structure type*)
		IsPowered : BOOL; (*True if powered*)
		IsHomed : BOOL; (*Status variable true if it is homed*)
		Error : BOOL; (*True if there is an error present*)
		MoveActive : BOOL; (*Checking if move is active*)
	END_STRUCT;
END_TYPE
```

### ConveyorIF.var - Conveyor interface varaibles
```iecst
(*global interface variables*)
VAR
	ConveyorController : ConveyorType; (*Conveyor control structure*)
END_VAR
```

### Program Logical/Source/Conveyor/Conveyor (IEC) - Sorting conveyor

#### Cyclic.ld - Cyclic code
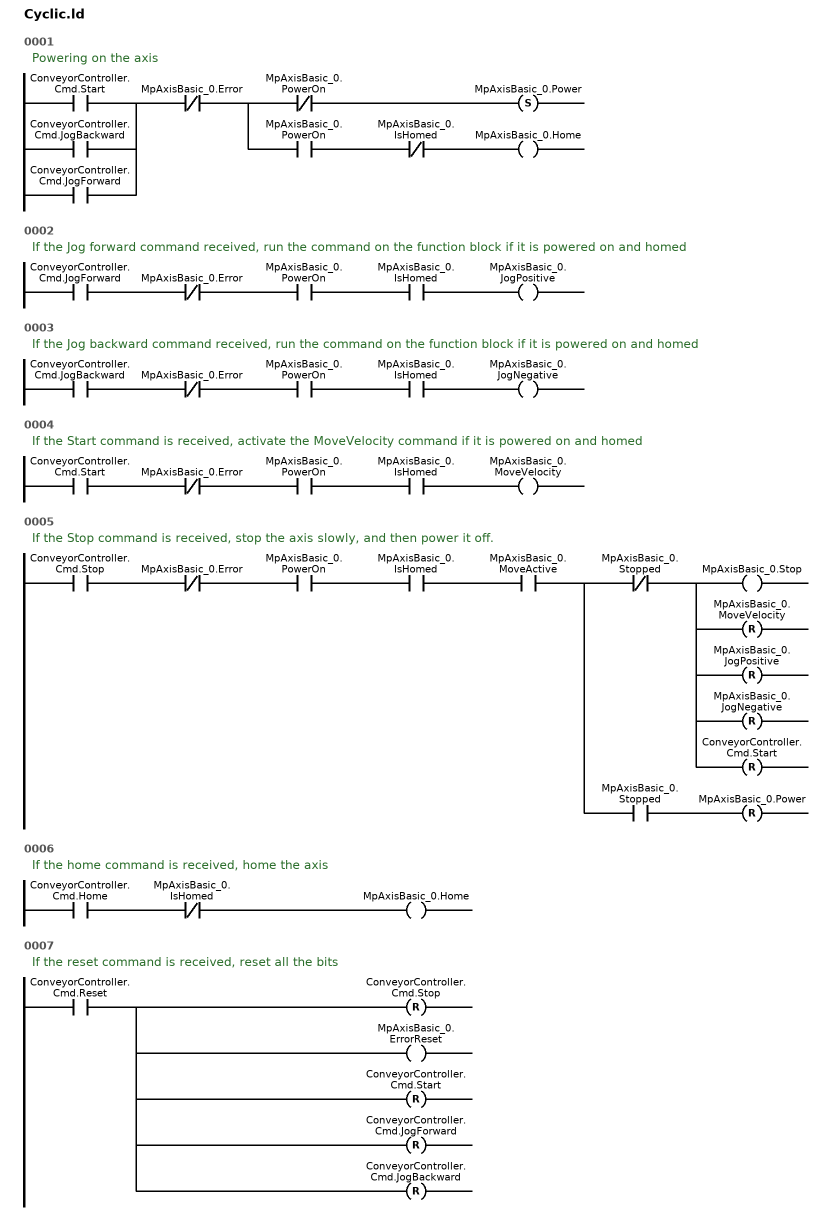
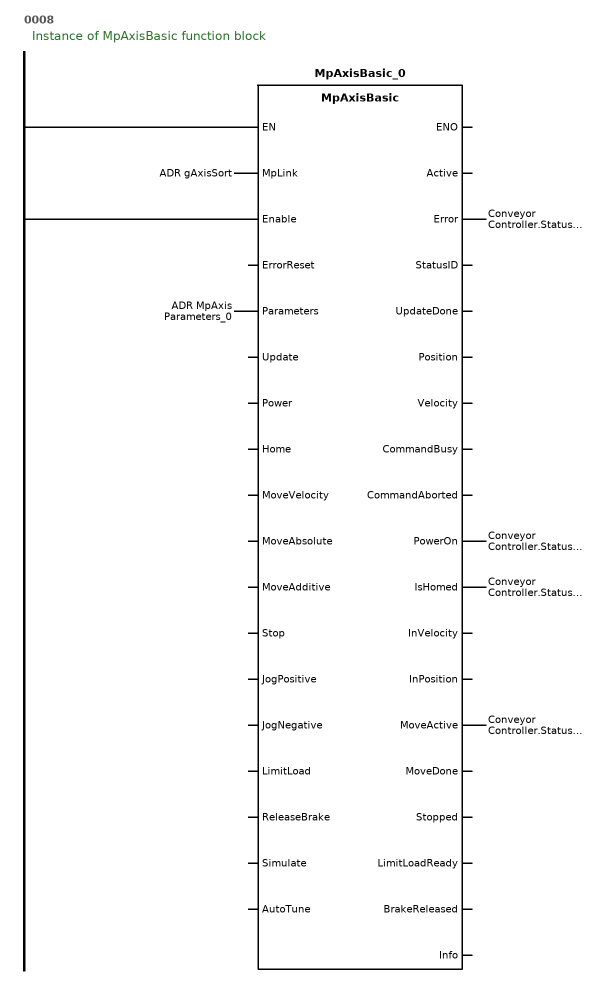
Ladder, written as Structured Text:
```iecst
PROGRAM _CYCLIC
VAR
    _p1 : BOOL;
    _p2 : BOOL;
    _p3 : BOOL;
    _p4 : BOOL;
END_VAR
(* Network 1: Powering on the axis *)
_p1 := (ConveyorController.Cmd.Start OR ConveyorController.Cmd.JogBackward OR ConveyorController.Cmd.JogForward) AND NOT MpAxisBasic_0.Error;
IF _p1 AND NOT MpAxisBasic_0.PowerOn THEN MpAxisBasic_0.Power := TRUE; END_IF;
MpAxisBasic_0.Home := _p1 AND MpAxisBasic_0.PowerOn AND NOT MpAxisBasic_0.IsHomed;

(* Network 2: If the Jog forward command received, run the command on the function block if it is powered on and homed *)
MpAxisBasic_0.JogPositive := ConveyorController.Cmd.JogForward AND NOT MpAxisBasic_0.Error AND MpAxisBasic_0.PowerOn AND MpAxisBasic_0.IsHomed;

(* Network 3: If the Jog backward command received, run the command on the function block if it is powered on and homed *)
MpAxisBasic_0.JogNegative := ConveyorController.Cmd.JogBackward AND NOT MpAxisBasic_0.Error AND MpAxisBasic_0.PowerOn AND MpAxisBasic_0.IsHomed;

(* Network 4: If the Start command is received, activate the MoveVelocity command if it is powered on and homed *)
MpAxisBasic_0.MoveVelocity := ConveyorController.Cmd.Start AND NOT MpAxisBasic_0.Error AND MpAxisBasic_0.PowerOn AND MpAxisBasic_0.IsHomed;

(* Network 5: If the Stop command is received, stop the axis slowly, and then power it off. *)
_p2 := ConveyorController.Cmd.Stop AND NOT MpAxisBasic_0.Error AND MpAxisBasic_0.PowerOn AND MpAxisBasic_0.IsHomed AND MpAxisBasic_0.MoveActive;
_p3 := _p2 AND NOT MpAxisBasic_0.Stopped;
MpAxisBasic_0.Stop := _p2 AND NOT MpAxisBasic_0.Stopped;
IF _p3 THEN
    MpAxisBasic_0.MoveVelocity := FALSE;
    MpAxisBasic_0.JogPositive := FALSE;
    MpAxisBasic_0.JogNegative := FALSE;
    ConveyorController.Cmd.Start := FALSE;
END_IF;
IF _p2 AND MpAxisBasic_0.Stopped THEN MpAxisBasic_0.Power := FALSE; END_IF;

(* Network 6: If the home command is received, home the axis *)
MpAxisBasic_0.Home := ConveyorController.Cmd.Home AND NOT MpAxisBasic_0.IsHomed;

(* Network 7: If the reset command is received, reset all the bits *)
_p4 := ConveyorController.Cmd.Reset;
IF ConveyorController.Cmd.Reset THEN ConveyorController.Cmd.Stop := FALSE; END_IF;
MpAxisBasic_0.ErrorReset := _p4;
IF _p4 THEN
    ConveyorController.Cmd.Start := FALSE;
    ConveyorController.Cmd.JogForward := FALSE;
    ConveyorController.Cmd.JogBackward := FALSE;
END_IF;

(* Network 8: Instance of MpAxisBasic function block *)
MpAxisBasic_0(MpLink := ADR(gAxisSort), Enable := TRUE, Parameters := ADR(MpAxisParameters_0));
ConveyorController.Status.Error := MpAxisBasic_0.Error;
ConveyorController.Status.IsPowered := MpAxisBasic_0.PowerOn;
ConveyorController.Status.IsHomed := MpAxisBasic_0.IsHomed;
ConveyorController.Status.MoveActive := MpAxisBasic_0.MoveActive;
END_PROGRAM
```

#### Init.ld - Initialization code
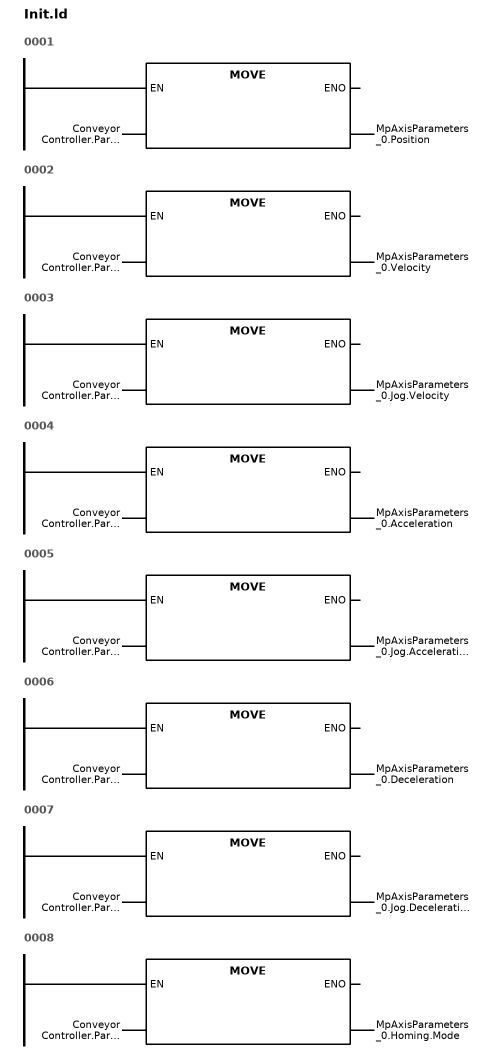
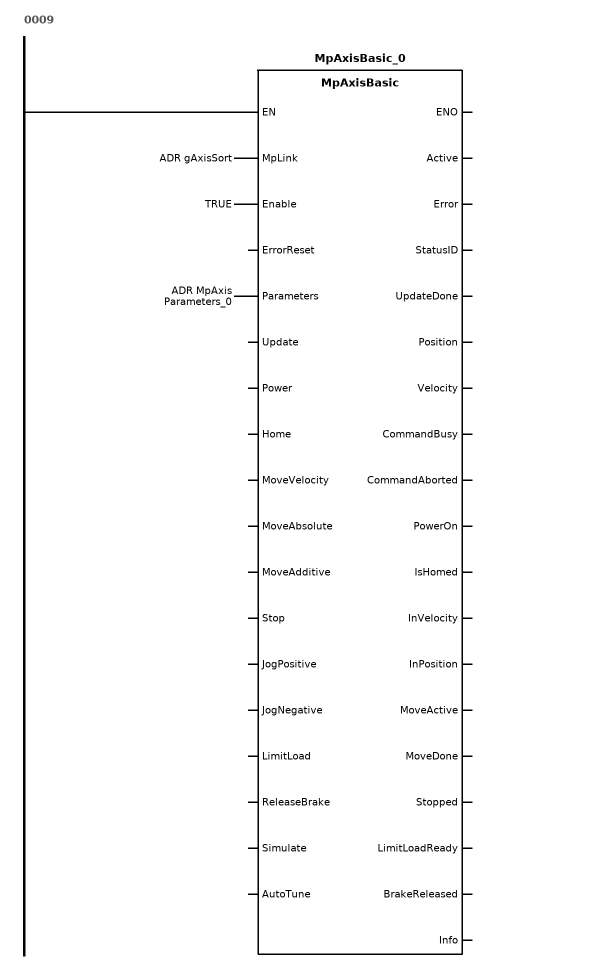
Ladder, written as Structured Text:
```iecst
PROGRAM _INIT
(* Network 1 *)
MpAxisParameters_0.Position := ConveyorController.Par.Position;

(* Network 2 *)
MpAxisParameters_0.Velocity := ConveyorController.Par.Velocity;

(* Network 3 *)
MpAxisParameters_0.Jog.Velocity := ConveyorController.Par.Velocity;

(* Network 4 *)
MpAxisParameters_0.Acceleration := ConveyorController.Par.Acceleration;

(* Network 5 *)
MpAxisParameters_0.Jog.Acceleration := ConveyorController.Par.Acceleration;

(* Network 6 *)
MpAxisParameters_0.Deceleration := ConveyorController.Par.Deceleration;

(* Network 7 *)
MpAxisParameters_0.Jog.Deceleration := ConveyorController.Par.Deceleration;

(* Network 8 *)
MpAxisParameters_0.Homing.Mode := ConveyorController.Par.HomingMode;

(* Network 9 *)
MpAxisBasic_0(MpLink := ADR(gAxisSort), Enable := TRUE, Parameters := ADR(MpAxisParameters_0));
END_PROGRAM
```

#### Exit.ld - Exit code
Ladder, written as Structured Text:
```iecst
PROGRAM _EXIT
END_PROGRAM
```

#### Types.typ - Local data types
```iecst
(*local enumerated types*)

TYPE
	MotionControlEnum :
		( (*Enum type for state machine variable*)
		mcINIT := 1, (*Intial state*)
		mcPOWER := 2, (*Powering on*)
		mcHOME := 3, (*Homing the axis*)
		mcWAIT_FOR_CMD := 4, (*Waiting for a move command*)
		mcPROCESS := 6, (*Process the move command*)
		mcERROR := 7 (*Error handling*)
		);
END_TYPE
```

#### Variables.var - Local variables
```iecst
(*local function blocks*)
VAR
	MpAxisBasic_0 : MpAxisBasic; (*MpAxisBasic function block to control stepper motor*)
END_VAR
(*local structures*)
VAR
	MpAxisParameters_0 : MpAxisBasicParType; (*Parameter structure for the axis*)
END_VAR
(*local enumerators*)
VAR
	MotionControlState : MotionControlEnum := mcINIT; (*Enumerator to keep track of state machine status*)
END_VAR
```

### Package Logical/Source/Sorter - Package for sorter source code

### SorterIF.typ - Interface types for Sorter
```iecst
(*global sorter interface types*)

TYPE
	SorterCommandType : 	STRUCT  (*Commands to pass to the sorter*)
		ExtendSwitch1 : BOOL; (*Command to extend the first switch*)
		ExtendSwitch2 : BOOL; (*Command to extend the second switch*)
		RetractStopper : BOOL; (*Command to retract the stopper*)
		InternalHome : BOOL; (*Separate command to home internally*)
		Home : BOOL; (*Command to home sorter*)
		Reset : BOOL; (*Command to reset*)
	END_STRUCT;
	SortingRecipeType : 	STRUCT  (*Recipe type for lane allocation*)
		Lane1ProductType : ProductTypeEnum; (*Lane 1 product type allocation*)
		Lane2ProductType : ProductTypeEnum; (*Lane 2 product type allocation*)
		Lane3ProductType : ProductTypeEnum; (*Lane 3 product type allocation*)
	END_STRUCT;
	SorterParameterType : 	STRUCT  (*Parameters for the sorter*)
		LaneAllocationRecipe : SortingRecipeType; (*Lane allocation recipe*)
	END_STRUCT;
	SorterErrors : 	STRUCT  (*Structure for the process errors of the sorter*)
		Error1 : BOOL; (*ERROR 1 = Cap not sorted, stuck on conveyor or ejected. Please check machine*)
		Error2 : BOOL; (*ERROR 2 = Cap stuck behind stopped*)
		Error3 : BOOL; (*ERROR 3 = One of the lanes is full*)
	END_STRUCT;
	SorterStates : 	STRUCT  (*Local state machine tracker*)
		Init : BOOL; (*Initial state*)
		InitDone : BOOL; (*Initial done bit*)
		Waiting : BOOL; (*Waiting state*)
		WaitingDone : BOOL; (*Waiting done bit*)
		Classifying : BOOL; (*Classifying state*)
		ClassifyingDone : BOOL; (*Classifying done bit*)
		SortingProduct : BOOL; (*Sorting state*)
		SortingProductDone : BOOL; (*Sorting done bit*)
		Error : BOOL; (*Error state*)
	END_STRUCT;
	SorterStatusType : 	STRUCT  (*Status variables from the sorter*)
		ProductAvailable : BOOL; (*Product is available at beginning of line*)
		ProductMetallic : BOOL; (*Product material sensor*)
		ProductNotBlack : BOOL; (*Product color sensor*)
		ProductType : ProductTypeEnum := ptUNKNOWN; (*Product type*)
		LaneFull : BOOL; (*Product in between stopper and sorting*)
		Switch1Retracted : BOOL; (*Switch 1 is retracted (not active)*)
		Switch1Extended : BOOL; (*Switch 1 is extended (active)*)
		Switch2Retracted : BOOL; (*Switch 2 is retracted (not active)*)
		Switch2Extended : BOOL; (*Switch 2 is extended (active)*)
		IsHomed : BOOL; (*True if all pneumatic valves in home position*)
		ProcessDone : BOOL; (*Process done bit*)
		SorterState : SorterStates; (*State machine local*)
		Errors : SorterErrors; (*Errors structure*)
		DestLane : UINT := 0; (*Destination lane, 1 2 or 3*)
	END_STRUCT;
	SorterType : 	STRUCT  (*Sorter custom type for interface*)
		Cmd : SorterCommandType; (*Command structure for sorter*)
		Par : SorterParameterType; (*Parameter structure for sorter*)
		Status : SorterStatusType; (*Status structure with feedback from sorter*)
	END_STRUCT;
	ProductCounterType : 	STRUCT  (*Product counter type*)
		ProductCountRed : UINT; (*Product counter for red products*)
		ProductCountBlack : UINT; (*Product counter for black products*)
		ProductCountMetal : UINT; (*Product counter for metal products*)
	END_STRUCT;
END_TYPE

(*global sorter enums*)

TYPE
	ProductTypeEnum :
		( (*Enumerator to track type of product*)
		ptUNKNOWN := 1, (*Initial state*)
		ptRED := 2, (*Product is red color and plastic*)
		ptBLACK := 3, (*Product is black color and plastic*)
		ptMETAL := 4 (*Product is metallic*)
		);
END_TYPE
```

### SorterIF.var - Interface variables for Sorter
```iecst
(*global sorter interface variables*)
VAR
	SorterControl : SorterType; (*Control structure for the Sorter*)
	ProductCounter : ProductCounterType; (*Counters for all three product types*)
END_VAR
```

### Program Logical/Source/Sorter/Sorter (IEC) - Sorter program

#### Cyclic.ld - Cyclic code
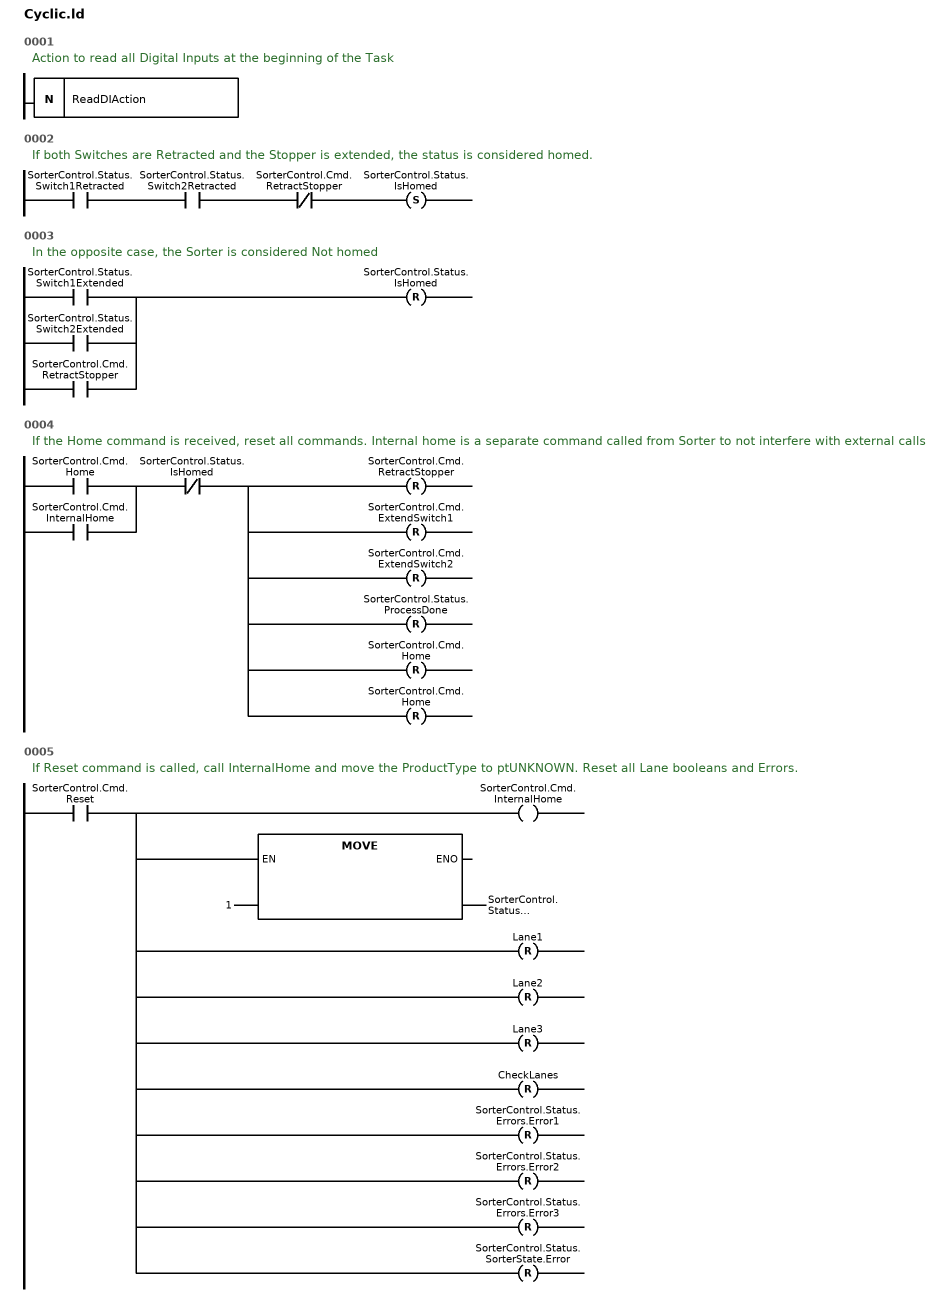
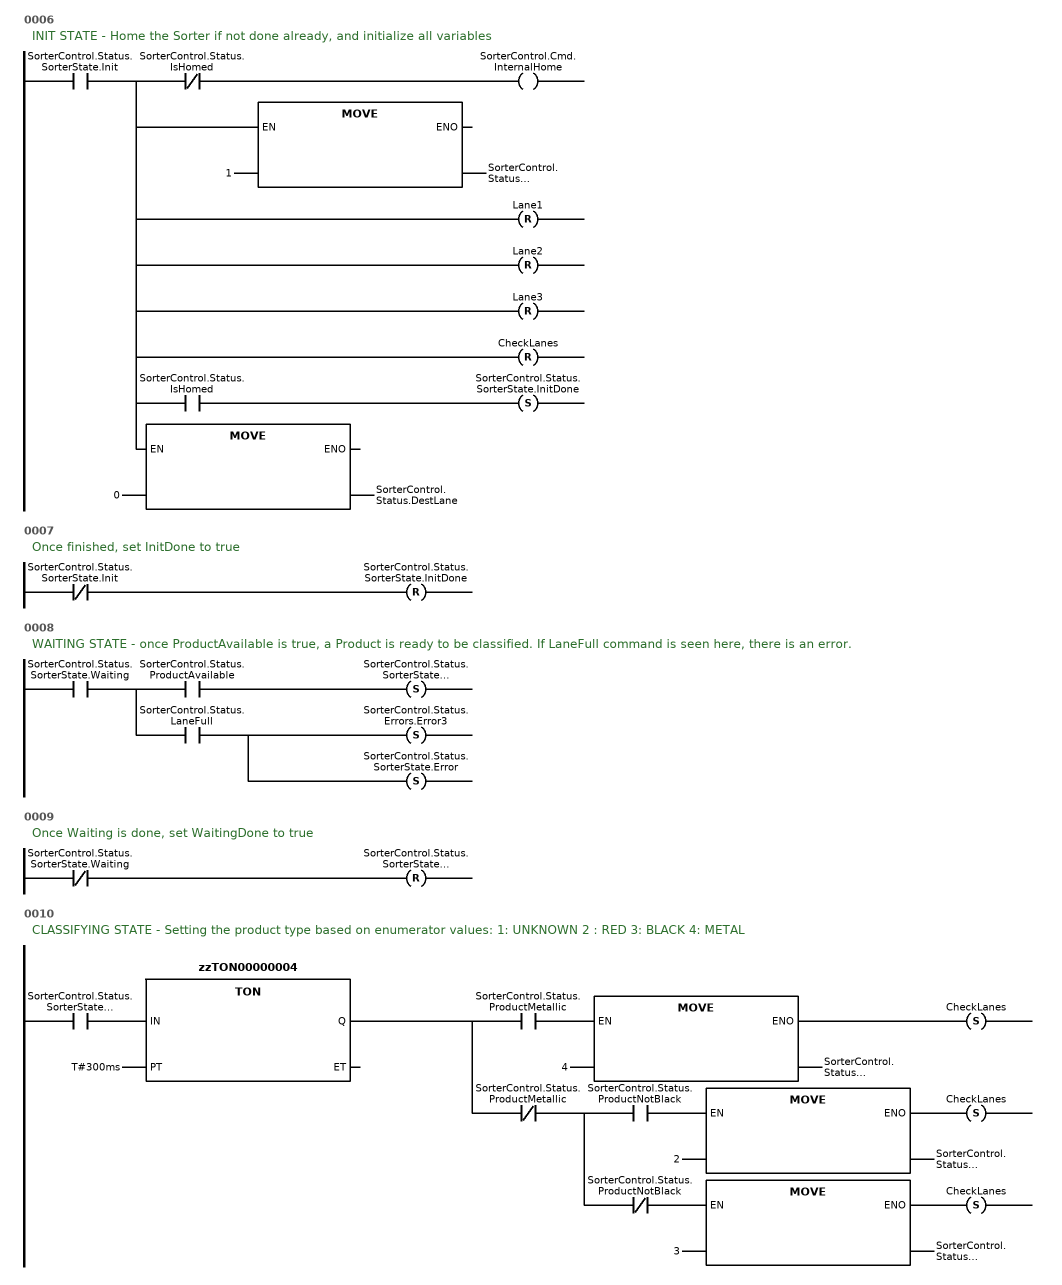
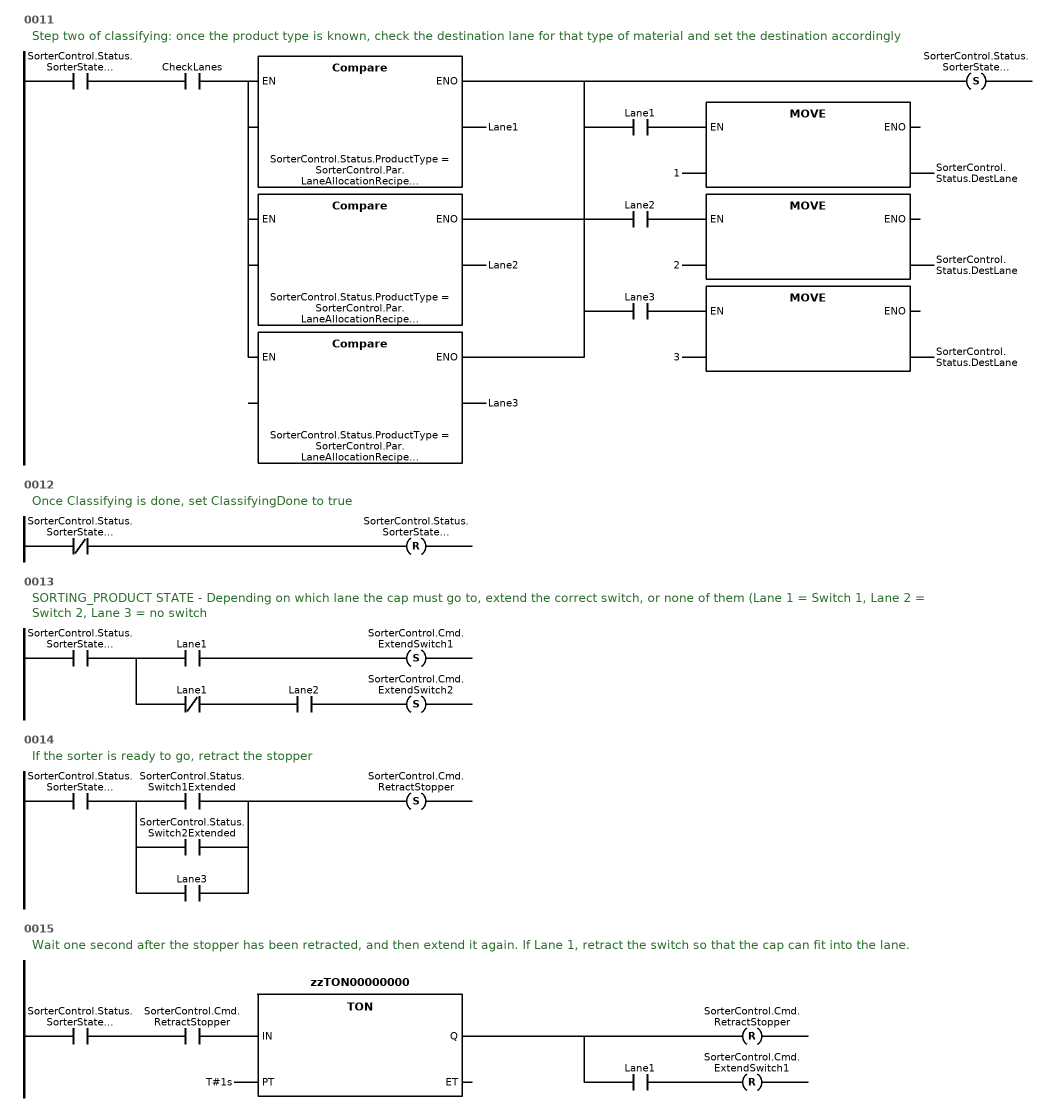
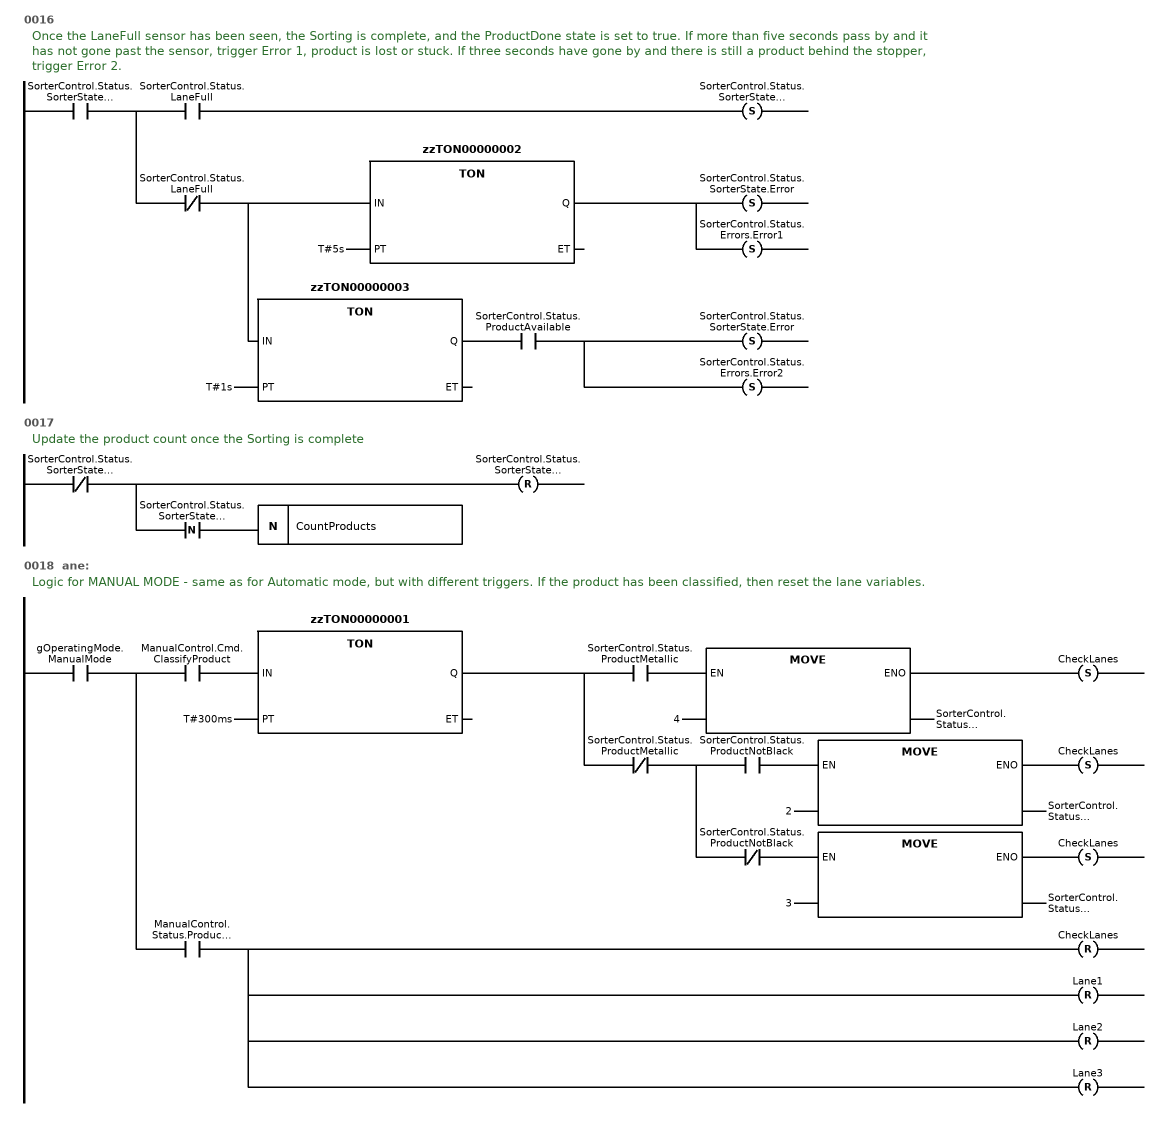
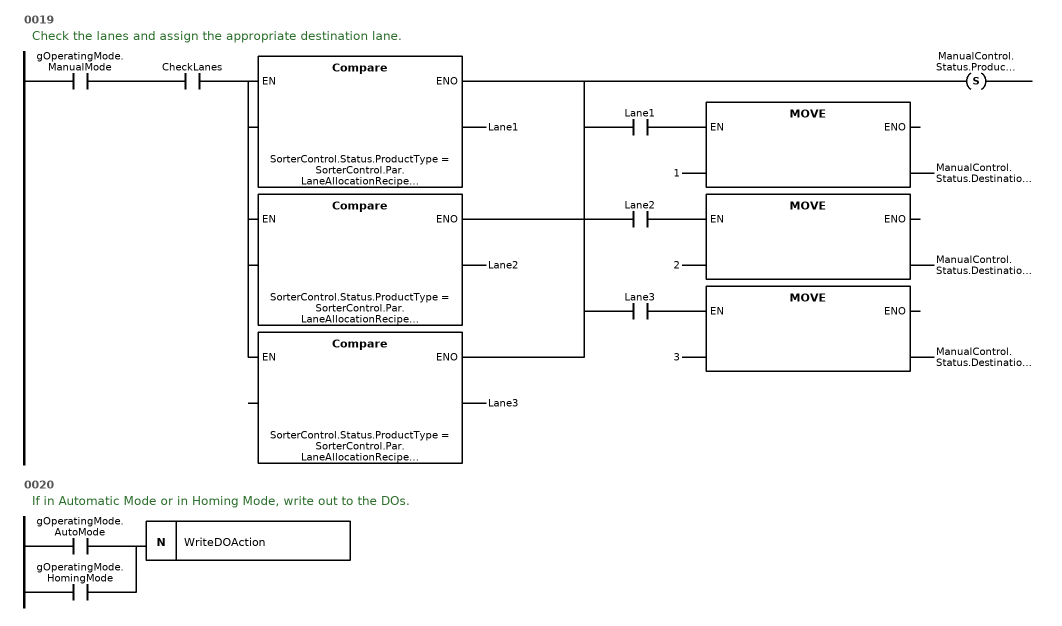
Ladder, written as Structured Text:
```iecst
PROGRAM _CYCLIC
VAR
    _p1 : BOOL;
    _p2 : BOOL;
    _p3 : BOOL;
    _p4 : BOOL;
    _p5 : BOOL;
    _p6 : BOOL;
    _p7 : BOOL;
    _p8 : BOOL;
    _p9 : BOOL;
    _p10 : BOOL;
    _p11 : BOOL;
    _p12 : BOOL;
    _p13 : BOOL;
    _p14 : BOOL;
    _p15 : BOOL;
    _e16 : F_TRIG;
    _p17 : BOOL;
    _p18 : BOOL;
    _p19 : BOOL;
    _p20 : BOOL;
    _p21 : BOOL;
END_VAR
(* Network 1: Action to read all Digital Inputs at the beginning of the Task *)
ReadDIAction;

(* Network 2: If both Switches are Retracted and the Stopper is extended, the status is considered homed. *)
IF SorterControl.Status.Switch1Retracted AND SorterControl.Status.Switch2Retracted AND NOT SorterControl.Cmd.RetractStopper THEN
    SorterControl.Status.IsHomed := TRUE;
END_IF;

(* Network 3: In the opposite case, the Sorter is considered Not homed *)
IF SorterControl.Status.Switch1Extended OR SorterControl.Status.Switch2Extended OR SorterControl.Cmd.RetractStopper THEN
    SorterControl.Status.IsHomed := FALSE;
END_IF;

(* Network 4: If the Home command is received, reset all commands. Internal home is a separate command called from Sorter to not interfere with external calls *)
_p1 := (SorterControl.Cmd.Home OR SorterControl.Cmd.InternalHome) AND NOT SorterControl.Status.IsHomed;
IF _p1 THEN
    SorterControl.Cmd.RetractStopper := FALSE;
    SorterControl.Cmd.ExtendSwitch1 := FALSE;
    SorterControl.Cmd.ExtendSwitch2 := FALSE;
    SorterControl.Status.ProcessDone := FALSE;
    SorterControl.Cmd.Home := FALSE;
    SorterControl.Cmd.Home := FALSE;
END_IF;

(* Network 5: If Reset command is called, call InternalHome and move the ProductType to ptUNKNOWN. Reset all Lane booleans and Errors. *)
_p2 := SorterControl.Cmd.Reset;
SorterControl.Cmd.InternalHome := SorterControl.Cmd.Reset;
IF _p2 THEN
    SorterControl.Status.ProductType := 1;
    Lane1 := FALSE;
    Lane2 := FALSE;
    Lane3 := FALSE;
    CheckLanes := FALSE;
    SorterControl.Status.Errors.Error1 := FALSE;
    SorterControl.Status.Errors.Error2 := FALSE;
    SorterControl.Status.Errors.Error3 := FALSE;
    SorterControl.Status.SorterState.Error := FALSE;
END_IF;

(* Network 6: INIT STATE - Home the Sorter if not done already, and initialize all variables *)
_p3 := SorterControl.Status.SorterState.Init;
SorterControl.Cmd.InternalHome := SorterControl.Status.SorterState.Init AND NOT SorterControl.Status.IsHomed;
IF _p3 THEN
    SorterControl.Status.ProductType := 1;
    Lane1 := FALSE;
    Lane2 := FALSE;
    Lane3 := FALSE;
    CheckLanes := FALSE;
END_IF;
IF _p3 AND SorterControl.Status.IsHomed THEN SorterControl.Status.SorterState.InitDone := TRUE; END_IF;
IF _p3 THEN SorterControl.Status.DestLane := 0; END_IF;

(* Network 7: Once finished, set InitDone to true *)
IF NOT SorterControl.Status.SorterState.Init THEN
    SorterControl.Status.SorterState.InitDone := FALSE;
END_IF;

(* Network 8: WAITING STATE - once ProductAvailable is true, a Product is ready to be classified. If LaneFull command is seen here, there is an error. *)
_p4 := SorterControl.Status.SorterState.Waiting;
IF SorterControl.Status.SorterState.Waiting AND SorterControl.Status.ProductAvailable THEN
    SorterControl.Status.SorterState.WaitingDone := TRUE;
END_IF;
_p5 := _p4 AND SorterControl.Status.LaneFull;
IF _p4 AND SorterControl.Status.LaneFull THEN SorterControl.Status.Errors.Error3 := TRUE; END_IF;
IF _p5 THEN SorterControl.Status.SorterState.Error := TRUE; END_IF;

(* Network 9: Once Waiting is done, set WaitingDone to true *)
IF NOT SorterControl.Status.SorterState.Waiting THEN
    SorterControl.Status.SorterState.WaitingDone := FALSE;
END_IF;

(* Network 10: CLASSIFYING STATE - Setting the product type based on enumerator values: 1: UNKNOWN 2 : RED 3: BLACK 4: METAL *)
zzTON00000004(IN := SorterControl.Status.SorterState.Classifying, PT := T#300ms);
_p6 := zzTON00000004.Q AND SorterControl.Status.ProductMetallic;
IF _p6 THEN
    SorterControl.Status.ProductType := 4;
    CheckLanes := TRUE;
END_IF;
_p7 := zzTON00000004.Q AND NOT SorterControl.Status.ProductMetallic;
_p8 := _p7 AND SorterControl.Status.ProductNotBlack;
IF _p8 THEN
    SorterControl.Status.ProductType := 2;
    CheckLanes := TRUE;
END_IF;
_p9 := _p7 AND NOT SorterControl.Status.ProductNotBlack;
IF _p9 THEN
    SorterControl.Status.ProductType := 3;
    CheckLanes := TRUE;
END_IF;

(* Network 11: Step two of classifying: once the product type is known, check the destination lane for that type of material and set the destination accordingly *)
_p10 := SorterControl.Status.SorterState.Classifying AND CheckLanes;
IF _p10 THEN
    Lane1 := SorterControl.Status.ProductType = SorterControl.Par.LaneAllocationRecipe.Lane1ProductType;
    Lane2 := SorterControl.Status.ProductType = SorterControl.Par.LaneAllocationRecipe.Lane2ProductType;
    Lane3 := SorterControl.Status.ProductType = SorterControl.Par.LaneAllocationRecipe.Lane3ProductType;
    SorterControl.Status.SorterState.ClassifyingDone := TRUE;
END_IF;
IF _p10 AND Lane1 THEN SorterControl.Status.DestLane := 1; END_IF;
IF _p10 AND Lane2 THEN SorterControl.Status.DestLane := 2; END_IF;
IF _p10 AND Lane3 THEN SorterControl.Status.DestLane := 3; END_IF;

(* Network 12: Once Classifying is done, set ClassifyingDone to true *)
IF NOT SorterControl.Status.SorterState.Classifying THEN
    SorterControl.Status.SorterState.ClassifyingDone := FALSE;
END_IF;

(* Network 13: SORTING_PRODUCT STATE - Depending on which lane the cap must go to, extend the correct switch, or none of them (Lane 1 = Switch 1, Lane 2 = Switch 2, Lane 3 = no switch *)
_p11 := SorterControl.Status.SorterState.SortingProduct;
IF SorterControl.Status.SorterState.SortingProduct AND Lane1 THEN
    SorterControl.Cmd.ExtendSwitch1 := TRUE;
END_IF;
IF _p11 AND NOT Lane1 AND Lane2 THEN SorterControl.Cmd.ExtendSwitch2 := TRUE; END_IF;

(* Network 14: If the sorter is ready to go, retract the stopper *)
IF SorterControl.Status.SorterState.SortingProduct AND (SorterControl.Status.Switch1Extended OR SorterControl.Status.Switch2Extended OR Lane3) THEN
    SorterControl.Cmd.RetractStopper := TRUE;
END_IF;

(* Network 15: Wait one second after the stopper has been retracted, and then extend it again. If Lane 1, retract the switch so that the cap can fit into the lane. *)
zzTON00000000(IN := SorterControl.Status.SorterState.SortingProduct AND SorterControl.Cmd.RetractStopper, PT := T#1s);
IF zzTON00000000.Q THEN SorterControl.Cmd.RetractStopper := FALSE; END_IF;
IF zzTON00000000.Q AND Lane1 THEN SorterControl.Cmd.ExtendSwitch1 := FALSE; END_IF;

(* Network 16: Once the LaneFull sensor has been seen, the Sorting is complete, and the ProductDone state is set to true. If more than five seconds pass by and it has not gone past the sensor, trigger Error 1, product is lost or stuck. If three seconds have gone by and there is still a product behind the stopper, trigger Error 2. *)
_p12 := SorterControl.Status.SorterState.SortingProduct;
IF SorterControl.Status.SorterState.SortingProduct AND SorterControl.Status.LaneFull THEN
    SorterControl.Status.SorterState.SortingProductDone := TRUE;
END_IF;
zzTON00000002(IN := _p12 AND NOT SorterControl.Status.LaneFull, PT := T#5s);
_p13 := _p12 AND NOT SorterControl.Status.LaneFull;
IF zzTON00000002.Q THEN
    SorterControl.Status.SorterState.Error := TRUE;
    SorterControl.Status.Errors.Error1 := TRUE;
END_IF;
zzTON00000003(IN := _p13, PT := T#1s);
_p14 := zzTON00000003.Q AND SorterControl.Status.ProductAvailable;
IF _p14 THEN
    SorterControl.Status.SorterState.Error := TRUE;
    SorterControl.Status.Errors.Error2 := TRUE;
END_IF;

(* Network 17: Update the product count once the Sorting is complete *)
_p15 := NOT SorterControl.Status.SorterState.SortingProduct;
IF _p15 THEN SorterControl.Status.SorterState.SortingProductDone := FALSE; END_IF;
_e16(CLK := SorterControl.Status.SorterState.SortingProductDone);
IF _p15 AND _e16.Q THEN CountProducts; END_IF;

(* Network 18: Logic for MANUAL MODE - same as for Automatic mode, but with different triggers. If the product has been classified, then reset the lane variables. *)
ane:
zzTON00000001(IN := gOperatingMode.ManualMode AND ManualControl.Cmd.ClassifyProduct, PT := T#300ms);
_p17 := zzTON00000001.Q AND SorterControl.Status.ProductMetallic;
IF _p17 THEN
    SorterControl.Status.ProductType := 4;
    CheckLanes := TRUE;
END_IF;
_p18 := zzTON00000001.Q AND NOT SorterControl.Status.ProductMetallic;
_p19 := _p18 AND SorterControl.Status.ProductNotBlack;
IF _p19 THEN
    SorterControl.Status.ProductType := 2;
    CheckLanes := TRUE;
END_IF;
_p20 := _p18 AND NOT SorterControl.Status.ProductNotBlack;
IF _p20 THEN
    SorterControl.Status.ProductType := 3;
    CheckLanes := TRUE;
END_IF;
_p21 := gOperatingMode.ManualMode AND ManualControl.Status.ProductClassified;
IF _p21 THEN
    CheckLanes := FALSE;
    Lane1 := FALSE;
    Lane2 := FALSE;
    Lane3 := FALSE;
END_IF;

(* Network 19: Check the lanes and assign the appropriate destination lane. *)
IF gOperatingMode.ManualMode AND CheckLanes THEN
    Lane1 := SorterControl.Status.ProductType = SorterControl.Par.LaneAllocationRecipe.Lane1ProductType;
    Lane2 := SorterControl.Status.ProductType = SorterControl.Par.LaneAllocationRecipe.Lane2ProductType;
    Lane3 := SorterControl.Status.ProductType = SorterControl.Par.LaneAllocationRecipe.Lane3ProductType;
    ManualControl.Status.ProductClassified := TRUE;
END_IF;
IF gOperatingMode.ManualMode AND CheckLanes AND Lane1 THEN
    ManualControl.Status.DestinationLane := 1;
END_IF;
IF gOperatingMode.ManualMode AND CheckLanes AND Lane2 THEN
    ManualControl.Status.DestinationLane := 2;
END_IF;
IF gOperatingMode.ManualMode AND CheckLanes AND Lane3 THEN
    ManualControl.Status.DestinationLane := 3;
END_IF;

(* Network 20: If in Automatic Mode or in Homing Mode, write out to the DOs. *)
IF gOperatingMode.AutoMode OR gOperatingMode.HomingMode THEN WriteDOAction; END_IF;
END_PROGRAM
```

#### Init.ld - Initialization code
Ladder, written as Structured Text:
```iecst
PROGRAM _INIT
END_PROGRAM
```

#### Exit.ld - Exit code
Ladder, written as Structured Text:
```iecst
PROGRAM _EXIT
END_PROGRAM
```

#### ReadDIAction.ld - Action file to read digital inputs from sorter
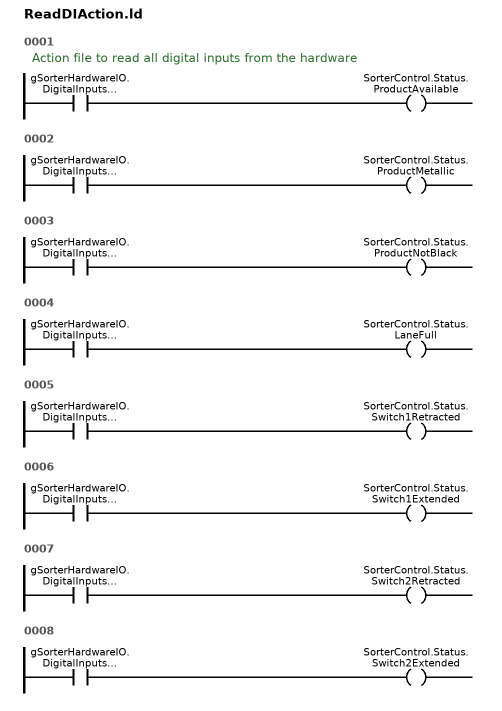
Ladder, written as Structured Text:
```iecst
ACTION ReadDIAction:
(* Network 1: Action file to read all digital inputs from the hardware *)
SorterControl.Status.ProductAvailable := gSorterHardwareIO.DigitalInputs.diProdAvail;

(* Network 2 *)
SorterControl.Status.ProductMetallic := gSorterHardwareIO.DigitalInputs.diMetallic;

(* Network 3 *)
SorterControl.Status.ProductNotBlack := gSorterHardwareIO.DigitalInputs.diNotBlack;

(* Network 4 *)
SorterControl.Status.LaneFull := gSorterHardwareIO.DigitalInputs.diLaneFull;

(* Network 5 *)
SorterControl.Status.Switch1Retracted := gSorterHardwareIO.DigitalInputs.diSwitch1Retracted;

(* Network 6 *)
SorterControl.Status.Switch1Extended := gSorterHardwareIO.DigitalInputs.diSwitch1Extended;

(* Network 7 *)
SorterControl.Status.Switch2Retracted := gSorterHardwareIO.DigitalInputs.diSwitch2Retracted;

(* Network 8 *)
SorterControl.Status.Switch2Extended := gSorterHardwareIO.DigitalInputs.diSwitch2Extended;
END_ACTION
```

#### WriteDOAction.ld - Action file to write digital outputs to sorter hardware
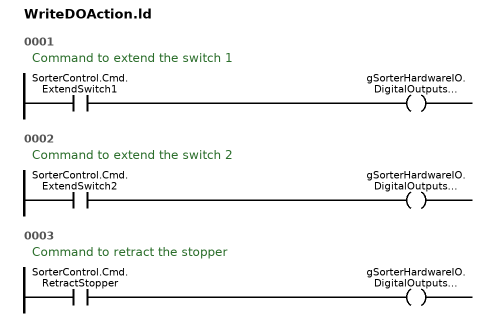
Ladder, written as Structured Text:
```iecst
ACTION WriteDOAction:
(* Network 1: Command to extend the switch 1 *)
gSorterHardwareIO.DigitalOutputs.doExtendSwitch1 := SorterControl.Cmd.ExtendSwitch1;

(* Network 2: Command to extend the switch 2 *)
gSorterHardwareIO.DigitalOutputs.doExtendSwitch2 := SorterControl.Cmd.ExtendSwitch2;

(* Network 3: Command to retract the stopper *)
gSorterHardwareIO.DigitalOutputs.doRetractStopper := SorterControl.Cmd.RetractStopper;
END_ACTION
```

#### CountProducts.ld - Action to count products
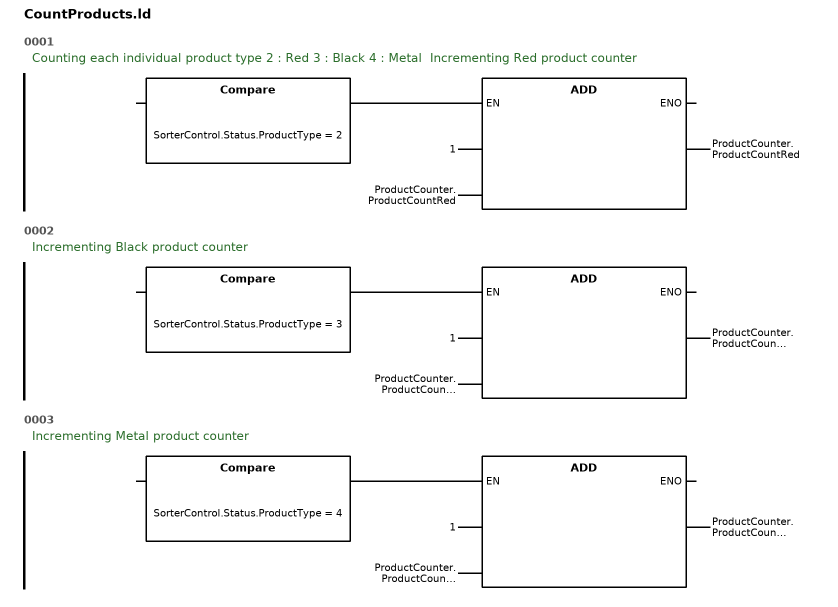
Ladder, written as Structured Text:
```iecst
ACTION CountProducts:
(* Network 1: Counting each individual product type 2 : Red 3 : Black 4 : Metal  Incrementing Red product counter *)
IF (SorterControl.Status.ProductType = 2) THEN
    ProductCounter.ProductCountRed := 1 + ProductCounter.ProductCountRed;
END_IF;

(* Network 2: Incrementing Black product counter *)
IF (SorterControl.Status.ProductType = 3) THEN
    ProductCounter.ProductCountBlack := 1 + ProductCounter.ProductCountBlack;
END_IF;

(* Network 3: Incrementing Metal product counter *)
IF (SorterControl.Status.ProductType = 4) THEN
    ProductCounter.ProductCountMetal := 1 + ProductCounter.ProductCountMetal;
END_IF;
END_ACTION
```

#### Variables.var - Local variables
```iecst
(*local variables*)
VAR
	Lane1 : BOOL; (*True if lane 1 is target*)
	Lane2 : BOOL; (*True if lane 2 is target*)
	Lane3 : BOOL; (*True if lane 3 is target*)
	CheckLanes : BOOL; (*Variable to activate action*)
END_VAR
```

### Package Logical/Infrastructure - Package for infrastructure code

### Package Logical/Infrastructure/Alarms - Package for MpAlarmX system

### Program Logical/Infrastructure/Alarms/AlarmHandling (IEC) - Alarms program

#### Main.st - Init, cyclic, exit code
```iecst
(*********************************************************************************
 * Copyright:   B&R Industrial Automation GmbH
 * Author:      lauryr
 * Created:     May 17, 2025/4:42 PM
 * Description: Structure text program implementing simple alarm handling
 *********************************************************************************)

PROGRAM _INIT

	// Enabling MpAlarmXCore function block
	MpAlarmXCore_0.Enable := TRUE;
	MpAlarmXCore_0.MpLink := ADR(MpLinkSORTING_gAlarmXCore);

	// Enabling MpAlarmXHistory function block
	MpAlarmXHistory_0.Enable := TRUE;
	MpAlarmXHistory_0.MpLink := ADR(MpLinkSORTING_gAlarmXHistory);

	// Enabling MpAlarmXAcknowledgeAll function block
	MpAlarmXAcknowledgeAll_0.Enable := TRUE;
	MpAlarmXAcknowledgeAll_0.MpLink := ADR(MpLinkSORTING_gAlarmXCore);

END_PROGRAM

PROGRAM _CYCLIC

	CommsErrors.X2X.X2X_ModuleOk := CommsErrors.X2X.X20BC0083_ModuleOk AND CommsErrors.X2X.X20BT9100_ModuleOk AND
		CommsErrors.X2X.X20DI9371_ModuleOk AND CommsErrors.X2X.X20DO9322_ModuleOk AND CommsErrors.X2X.X20PD0011_ModuleOk
		AND CommsErrors.X2X.X20PD0012_ModuleOk AND CommsErrors.X2X.X20PS9400_ModuleOk AND CommsErrors.X2X.X67SM2436_ModuleOk;

	// Automatic module errors - 1000 range
	IF AutomaticController.Status.Errors.Error1 THEN
	 	MpAlarmXSet(MpLinkSORTING_gAlarmXCore, 'Sorting station not homed');
 	ELSE
 		MpAlarmXReset(MpLinkSORTING_gAlarmXCore, 'Sorting station not homed');
	END_IF

	// Sorter module errors - 2000 range
	IF SorterControl.Status.Errors.Error1 THEN
		MpAlarmXSet(MpLinkSORTING_gAlarmXCore, 'Product stuck between stopper and lane');
	ELSE
		MpAlarmXReset(MpLinkSORTING_gAlarmXCore, 'Product stuck between stopper and lane');
	END_IF

	IF SorterControl.Status.Errors.Error2 THEN
		MpAlarmXSet(MpLinkSORTING_gAlarmXCore, 'Product behind stopper');
	ELSE
		MpAlarmXReset(MpLinkSORTING_gAlarmXCore, 'Product behind stopper');
	END_IF

	// Manual module errors - 3000 range
	IF ManualControl.Status.Error THEN
		MpAlarmXSet(MpLinkSORTING_gAlarmXCore, 'Incorrect switch open');
	ELSE
		MpAlarmXReset(MpLinkSORTING_gAlarmXCore, 'Incorrect switch open');
	END_IF

	// Comms errors - 4000 range
	IF NOT CommsErrors.PLK.FPLK_ModuleOk THEN
		MpAlarmXSet(MpLinkSORTING_gAlarmXCore, 'PLK comms error');
	ELSE
		MpAlarmXReset(MpLinkSORTING_gAlarmXCore, 'PLK comms error');
	END_IF

	IF NOT CommsErrors.X2X.X2X_ModuleOk THEN
		MpAlarmXSet(MpLinkSORTING_gAlarmXCore, 'X2X comms error');
	ELSE
		MpAlarmXReset(MpLinkSORTING_gAlarmXCore, 'X2X comms error');
	END_IF

	// Calling all function blocks cyclically
	MpAlarmXCore_0();
	MpAlarmXHistory_0();
	MpAlarmXAcknowledgeAll_0();

END_PROGRAM

PROGRAM _EXIT

	// Disabling MpAlarmXCore function block
	MpAlarmXCore_0.Enable := FALSE;
	MpAlarmXCore_0();

	// Disabling MpAlarmXHistory function block
	MpAlarmXHistory_0.Enable := FALSE;
	MpAlarmXHistory_0();

	// Disabling MpAlarmXAcknowledgeAll function block
	MpAlarmXAcknowledgeAll_0.Enable := FALSE;
	MpAlarmXAcknowledgeAll_0();

END_PROGRAM
```

#### Types.typ - Local data types
```iecst
(*local structure types*)

TYPE
	ErrorTypePLK : 	STRUCT  (*Structure to capture all PLK module errors*)
		FPLK_ModuleOk : BOOL; (*Powerlink card on the PPC2100*)
	END_STRUCT;
	ErrorTypeX2X : 	STRUCT  (*Structure to capture all X2X module errors*)
		X20BC0083_ModuleOk : BOOL; (*X2X bus controller communicating*)
		X20DI9371_ModuleOk : BOOL; (*Digital input module communicating*)
		X20PS9400_ModuleOk : BOOL; (*Power supply communicating*)
		X20PD0012_ModuleOk : BOOL; (*Potential distributor communicating*)
		X20PD0011_ModuleOk : BOOL; (*Potential distributor communicating*)
		X20DO9322_ModuleOk : BOOL; (*Digital output module communicating*)
		X20BT9100_ModuleOk : BOOL; (*Bus transmitter communicating*)
		X67SM2436_ModuleOk : BOOL; (*Stepper drive communicating*)
		X2X_ModuleOk : BOOL; (*General ok bit for X2X bus*)
	END_STRUCT;
	ErrorTypeComms : 	STRUCT  (*Structure to capture all errors in comms and of modules*)
		PLK : ErrorTypePLK; (*Powerlink errors*)
		X2X : ErrorTypeX2X; (*X2X errors*)
	END_STRUCT;
END_TYPE
```

#### Variables.var - Local variables
```iecst
(*local variables*)
VAR
	CommsErrors : ErrorTypeComms; (*Error structure for communications*)
END_VAR
(*local function blocks*)
VAR
	MpAlarmXAcknowledgeAll_0 : MpAlarmXAcknowledgeAll; (*MpAlarmXAcknowledgeAll function block*)
	MpAlarmXCore_0 : MpAlarmXCore; (*MpAlarmXCore function block*)
	MpAlarmXHistory_0 : MpAlarmXHistory; (*MpAlarmXHistory function block*)
END_VAR
```

### Package Logical/Infrastructure/Recipe - Package containing recipe implementation

### Program Logical/Infrastructure/Recipe/Recipe (IEC) - Recipe system

#### Main.st - Init, cyclic, exit code
```iecst
(*********************************************************************************
 * Copyright:   B&R Industrial Automation GmbH
 * Author:      lauryr
 * Created:     May 14, 2025/1:30 PM
 * Description: Recipe system to pick the lane allocation for different product types
 *********************************************************************************)

PROGRAM _INIT

	// Initialize MpRecipeXml function block
	MpRecipeXml_0.Enable := TRUE;
	MpRecipeXml_0.MpLink := ADR(MpLinkSORTING_gRecipeXml);
	MpRecipeXml_0.DeviceName := ADR('USER');
	// Initialize MpRecipeRegPar function block and assign PV
	MpRecipeRegPar_0.Enable := TRUE;
	MpRecipeRegPar_0.MpLink := ADR(MpLinkSORTING_gRecipeXml);
	MpRecipeRegPar_0.PVName := ADR('::SorterControl.Par.LaneAllocationRecipe');
	// Initialize MpRecipeUI function block
	MpRecipeUI_0.Enable := TRUE;
	MpRecipeUI_0.MpLink := ADR(MpLinkSORTING_gRecipeXml);
	MpRecipeUI_0.UIConnect := ADR(MpRecipeUIConnect);

END_PROGRAM

PROGRAM _CYCLIC

	// Calling selected value for use in other tasks
	selectedValue;
	// Call CreateRecipe action to create default recipe
	CreateRecipes;
	// Load default recipe into PV
	MpRecipeUIConnect.Recipe.Load;

	// Cyclically call all function blocks
	MpRecipeXml_0();
	MpRecipeRegPar_0();
	MpRecipeUI_0();

END_PROGRAM

PROGRAM _EXIT

	// Disable MpRecipeXml function block
	MpRecipeXml_0.Enable := FALSE;
	MpRecipeXml_0();
	// Disable MpRecipeRegPar function block
	MpRecipeRegPar_0.Enable := FALSE;
	MpRecipeRegPar_0();
	// Disable MpRecipeUI function block
	MpRecipeUI_0.Enable := FALSE;
	MpRecipeUI_0();

END_PROGRAM
```

#### CreateRecipes.st - Action file to create default recipe
```iecst
(*********************************************************************************
 * Copyright:   B&R Industrial Automation GmbH
 * Author:      lauryr
 * Created:     May 7, 2025/9:39 AM
 * Description: Action file to create default recipes
 *********************************************************************************)

ACTION CreateRecipes:

	// create default recipes in case they don't exist yet on the target
	// recipes are created by using the the MpRecipeXml instance interface

	CASE RecipeCreateStep OF
		IDLE:

			IF MpRecipeXml_0.Active = TRUE AND MpRecipeUI_0.Active = TRUE THEN

				// check for load error > triggers the default creation > if no error everything is ready to go
				IF (MpRecipeUIConnect.Recipe.List.Names[0] = '') THEN
					MpRecipeXml_0.Load 			:= FALSE;
					MpRecipeXml_0.ErrorReset 	:= TRUE;
					RecipeCreateStep 			:= CREATE_1;

				ELSE
					MpRecipeUIConnect.Recipe.Load := TRUE;
				END_IF

				// reset the load command from the init when recipe was loaded successfully
				IF (MpRecipeUIConnect.Status = mpRECIPE_UI_STATUS_LOAD) AND (MpRecipeUIConnect.Recipe.Load = TRUE) THEN
					MpRecipeUIConnect.Recipe.Load			:= FALSE;
					RecipeCreateStep						:= ALL_DONE;
				END_IF

			END_IF

		CREATE_1:	// Default recipe
			MpRecipeXml_0.ErrorReset 			:= FALSE;

			// Setting default values for RBM.xml
			SorterControl.Par.LaneAllocationRecipe.Lane1ProductType := ptRED;
			SorterControl.Par.LaneAllocationRecipe.Lane2ProductType := ptBLACK;
			SorterControl.Par.LaneAllocationRecipe.Lane3ProductType := ptMETAL;

			MpRecipeXml_0.FileName 				:= ADR(RECIPE_1_FILENAME);
			MpRecipeXml_0.Save					:= TRUE;
			RecipeCreateStep 					:= DONE_1;

		DONE_1:	// when CommandDone GoTo next step
			IF(MpRecipeXml_0.CommandDone) THEN
				RecipeCreateStep 			:= CREATE_2;
				MpRecipeXml_0.Save			:= FALSE;
			END_IF;

		CREATE_2:	// Default recipe
			MpRecipeXml_0.ErrorReset 			:= FALSE;

			// Setting default values for RMB.xml
			SorterControl.Par.LaneAllocationRecipe.Lane1ProductType := ptRED;
			SorterControl.Par.LaneAllocationRecipe.Lane2ProductType := ptMETAL;
			SorterControl.Par.LaneAllocationRecipe.Lane3ProductType := ptBLACK;

			MpRecipeXml_0.FileName 				:= ADR(RECIPE_2_FILENAME);
			MpRecipeXml_0.Save					:= TRUE;
			RecipeCreateStep 					:= DONE_2;

		DONE_2:	// when CommandDone GoTo next step
			IF(MpRecipeXml_0.CommandDone) THEN
				RecipeCreateStep 			:= CREATE_3;
				MpRecipeXml_0.Save			:= FALSE;
			END_IF;

		CREATE_3:	// Default recipe
			MpRecipeXml_0.ErrorReset 			:= FALSE;

			// Setting default values for BRM.xml
			SorterControl.Par.LaneAllocationRecipe.Lane1ProductType := ptBLACK;
			SorterControl.Par.LaneAllocationRecipe.Lane2ProductType := ptRED;
			SorterControl.Par.LaneAllocationRecipe.Lane3ProductType := ptMETAL;

			MpRecipeXml_0.FileName 				:= ADR(RECIPE_3_FILENAME);
			MpRecipeXml_0.Save					:= TRUE;
			RecipeCreateStep 					:= DONE_3;

		DONE_3:	// when CommandDone GoTo next step
			IF(MpRecipeXml_0.CommandDone) THEN
				RecipeCreateStep 			:= CREATE_4;
				MpRecipeXml_0.Save			:= FALSE;
			END_IF;

		CREATE_4:	// Default recipe
			MpRecipeXml_0.ErrorReset 			:= FALSE;

			// Setting default values for BMR.xml
			SorterControl.Par.LaneAllocationRecipe.Lane1ProductType := ptBLACK;
			SorterControl.Par.LaneAllocationRecipe.Lane2ProductType := ptMETAL;
			SorterControl.Par.LaneAllocationRecipe.Lane3ProductType := ptRED;

			MpRecipeXml_0.FileName 				:= ADR(RECIPE_4_FILENAME);
			MpRecipeXml_0.Save					:= TRUE;
			RecipeCreateStep 					:= DONE_4;

		DONE_4:	// when CommandDone GoTo next step
			IF(MpRecipeXml_0.CommandDone) THEN
				RecipeCreateStep 			:= CREATE_5;
				MpRecipeXml_0.Save			:= FALSE;
			END_IF;

		CREATE_5:	// Default recipe
			MpRecipeXml_0.ErrorReset 			:= FALSE;

			// Setting default values for BMR.xml
			SorterControl.Par.LaneAllocationRecipe.Lane1ProductType := ptMETAL;
			SorterControl.Par.LaneAllocationRecipe.Lane2ProductType := ptRED;
			SorterControl.Par.LaneAllocationRecipe.Lane3ProductType := ptBLACK;

			MpRecipeXml_0.FileName 				:= ADR(RECIPE_5_FILENAME);
			MpRecipeXml_0.Save					:= TRUE;
			RecipeCreateStep 					:= DONE_5;

		DONE_5:	// when CommandDone GoTo next step
			IF(MpRecipeXml_0.CommandDone) THEN
				RecipeCreateStep 			:= CREATE_6;
				MpRecipeXml_0.Save			:= FALSE;
			END_IF;

		CREATE_6:	// Default recipe
			MpRecipeXml_0.ErrorReset 			:= FALSE;

			// Setting default values for DefaultRecipe.xml
			SorterControl.Par.LaneAllocationRecipe.Lane1ProductType := ptMETAL;
			SorterControl.Par.LaneAllocationRecipe.Lane2ProductType := ptBLACK;
			SorterControl.Par.LaneAllocationRecipe.Lane3ProductType := ptRED;

			MpRecipeXml_0.FileName 				:= ADR(RECIPE_6_FILENAME);
			MpRecipeXml_0.Save					:= TRUE;
			RecipeCreateStep 					:= REFRESH;

		REFRESH:	// refresh the recipe list to make sure all the recipes are shown

			IF(MpRecipeXml_0.CommandDone) THEN
				RecipeCreateStep 					:= LOAD;
				MpRecipeXml_0.Save					:= FALSE;
				MpRecipeUIConnect.Recipe.Refresh 	:= TRUE;
			END_IF;

		LOAD:	// load the first recipe to have a default recipe

			IF(MpRecipeUIConnect.Status = mpRECIPE_UI_STATUS_IDLE)THEN
				MpRecipeUIConnect.Recipe.Load 		:= TRUE;
				RecipeCreateStep 					:= DONE_6;
			END_IF

		DONE_6:	// if loading was successful the creation of the recipes is done

			IF(MpRecipeUIConnect.Status = mpRECIPE_UI_STATUS_IDLE)THEN
				RecipeCreateStep 					:= ALL_DONE;
				MpRecipeUIConnect.Recipe.Refresh 	:= FALSE;
				MpRecipeUIConnect.Recipe.Load 		:= FALSE;
			END_IF;

	END_CASE;

END_ACTION
```

#### Types.typ - Local data types
```iecst
(*local recipe state machine type*)

TYPE
	RecipeCreateSteps :
		( (*Steps for creating recipes*)
		IDLE := 0, (*Idle State *)
		CREATE_1 := 10, (*Create first recipe*)
		DONE_1 := 11, (*First recipe done*)
		CREATE_2 := 20, (*Create second recipe*)
		DONE_2 := 21, (*Second recipe done*)
		CREATE_3 := 30, (*Create third recipe*)
		DONE_3 := 31, (*Third recipe done*)
		CREATE_4 := 40, (*Create fourth recipe*)
		DONE_4 := 41, (*Fourth recipe done*)
		CREATE_5 := 50, (*Create fifth recipe*)
		DONE_5 := 51, (*Fifth recipe done*)
		CREATE_6 := 60, (*Create sixth recipe*)
		DONE_6 := 61, (*Sixth recipe done*)
		REFRESH := 62, (*Reload the recipe object*)
		LOAD := 63, (*Load the recipe*)
		ALL_DONE := 70 (*All recipes were created*)
		);
END_TYPE
```

#### Variables.var - Local variables
```iecst
(*local variables*)
VAR
	SaveRecipe : BOOL := FALSE; (*Command to save recipes*)
	RecipeCreateStep : RecipeCreateSteps := IDLE; (*Internal variable for recipe creating state machine*)
	MpRecipeUIConnect : MpRecipeUIConnectType := (Recipe:=(Filter:='*xml'),New:=(FileName:='newRecipe.xml')); (*MpRecipeUI connection datapoints*)
	RecipeList : ARRAY[0..19] OF STRING[100] := ['{"value":"BMR.xml","text":"BMR.xml"}','{"value":"BRM.xml","text":"BRM.xml"}','{"value":"MBR.xml","text":"MBR.xml"}','{"value":"MRB.xml","text":"MRB.xml"}','{"value":"RBM.xml","text":"RBM.xml"}','{"value":"RMB.xml","text":"RMB.xml"}',14('')]; (*List box data provider*)
	selectedValue : STRING[100]; (*Selected value from list box*)
END_VAR
(*local function blocks*)
VAR
	MpRecipeRegPar_0 : MpRecipeRegPar; (*Registration of the recipe structure variable*)
	MpRecipeUI_0 : MpRecipeUI := (UISetup:=(RecipeListSize:=11,RecipeListScrollWindow:=0,Confirmation:=(RecipeLoad:=0,RecipeSave:=0,RecipeCreate:=0,RecipeDelete:=TRUE))); (*MpRecipeUI Component*)
	MpRecipeXml_0 : MpRecipeXml; (*Recipe Handling FUB*)
	LoadRecipe : BOOL; (*Load recipe*)
END_VAR
(*local constants*)
VAR
	RECIPE_6_FILENAME : STRING[255] := 'MBR.xml'; (*Metal Black Red recipe file name*)
	RECIPE_5_FILENAME : STRING[255] := 'MRB.xml'; (*Metal Red Black recipe file name*)
	RECIPE_4_FILENAME : STRING[255] := 'BMR.xml'; (*Black Metal Red recipe file name*)
	RECIPE_3_FILENAME : STRING[255] := 'BRM.xml'; (*Black Red Metal recipe file name*)
	RECIPE_2_FILENAME : STRING[255] := 'RMB.xml'; (*Red Metal Black recipe file name*)
	RECIPE_1_FILENAME : STRING[255] := 'RBM.xml'; (*Red Black Metal recipe file name*)
END_VAR
```

### Package Logical/Infrastructure/HMIHelper - Package containing HMI helper code

### HMIHelpIF.var - Interface variables for HMI helper
```iecst
VAR
	NewRecipeLoaded : BOOL;
END_VAR
```

### Program Logical/Infrastructure/HMIHelper/HMIHelper (IEC) - HMI helper task

#### Main.st - Init, cyclic, exit code
```iecst
(*********************************************************************************
 * Copyright:   B&R Industrial Automation GmbH
 * Author:      lauryr
 * Created:     May 17, 2025/5:10 PM
 * Description: HMI helper task to send and receive data to visualization and control
 *********************************************************************************)

PROGRAM _INIT

END_PROGRAM

PROGRAM _CYCLIC

	IF StopMode THEN
		AutomaticMode := FALSE;
		HomingMode := FALSE;
		ManualMode := FALSE;
		ActiveMode := 'Machine Stopped';
		IF NOT OpcUaControl.Read.DistributionReady THEN
			SortingStationStatus := 'Distribution Station error active';
		ELSE
			SortingStationStatus := 'Machine is stopped, select mode and press start';
		END_IF
	END_IF

	AutomaticController.Status.SortingReady := AutomaticMode OR OpcUaControl.Read.AutomaticActive;

	IF NewRecipeLoaded THEN
		SortingStationStatus := 'Please home the machine before starting automatic mode';
	END_IF

	IF AutomaticMode AND StartMode THEN
		HomingMode := FALSE;
		ManualMode := FALSE;
		ActiveMode := 'Automatic Mode';
		gOperatingMode.AutoMode := TRUE;
		gOperatingMode.HomingMode := FALSE;
		gOperatingMode.ManualMode := FALSE;
		ManualEnable := FALSE;
		SortingStationStatus := 'Automatic control active, normal operation';
		OpModeState := omAUTOMATIC;
		AutomaticActive := TRUE;
	ELSIF HomingMode AND StartMode THEN
		AutomaticActive := FALSE;
		AutomaticMode := FALSE;
		ManualMode := FALSE;
		ActiveMode := 'Homing Mode';
		gOperatingMode.HomingMode := TRUE;
		// Keeping automatic mode true to retain the state
		gOperatingMode.ManualMode := FALSE;
		ManualEnable := FALSE;
		OpModeState := omHOMING;
		SortingStationStatus := 'Please home the machine before starting automatic mode';
	ELSIF ManualMode AND StartMode THEN
		AutomaticActive := FALSE;
		AutomaticMode := FALSE;
		HomingMode := FALSE;
		ActiveMode := 'Manual Mode';
		gOperatingMode.ManualMode := TRUE;
		gOperatingMode.HomingMode := FALSE;
		gOperatingMode.AutoMode := FALSE;

		ManualEnable := TRUE;
		OpModeState := omMANUAL;

		SortingStationStatus := 'Manual control active, normal operation';
	END_IF

	CASE OpModeState OF
		omMANUAL:

			IF ManualControl.Status.Error THEN
				ErrorMessageManualPage := 'ERROR: Illegal movement, see guidelines';
				SortingStationStatus := 'Manual Mode Error - see Alarm page for more detail';
			ELSE
				ErrorMessageManualPage := 'Normal operation, no errors present';
				SortingStationStatus := 'Manual control active, normal operation';
			END_IF
			IF ManualControl.Status.DestinationLane = 1 THEN
				RequiredSwitch := 'Switch 1';
			ELSIF ManualControl.Status.DestinationLane = 2 THEN
				RequiredSwitch := 'Switch 2';
			ELSIF ManualControl.Status.DestinationLane = 3 THEN
				RequiredSwitch := 'None';
			ELSE
				RequiredSwitch := 'No product identified';
			END_IF

		omAUTOMATIC:
			IF SorterControl.Status.ProductType <> ptUNKNOWN THEN
				AutoIdentifiedProduct := TRUE;
			ELSE
				AutoIdentifiedProduct := FALSE;
			END_IF

			IF AutomaticController.Status.Errors.Error1 THEN
				SortingStationStatus := 'Automatic Mode Error - see Alarm page for more detail';
			ELSE
				SortingStationStatus := 'Automatic control active, normal operation';
			END_IF

		omHOMING:

	END_CASE

	IF SorterControl.Status.ProductType = ptRED THEN
		ProductRed := TRUE;
		ProductBlack := FALSE;
		ProductMetal := FALSE;
	ELSIF SorterControl.Status.ProductType = ptBLACK THEN
		ProductBlack := TRUE;
		ProductRed := FALSE;
		ProductMetal := FALSE;
	ELSIF SorterControl.Status.ProductType = ptMETAL THEN
		ProductMetal := TRUE;
		ProductRed := FALSE;
		ProductBlack := FALSE;
	ELSE
		ProductMetal := FALSE;
		ProductRed := FALSE;
		ProductBlack := FALSE;
	END_IF

	IF SorterControl.Par.LaneAllocationRecipe.Lane1ProductType = ptRED THEN
		RecipeItemLane1 := 'RED';
	ELSIF SorterControl.Par.LaneAllocationRecipe.Lane1ProductType = ptBLACK THEN
		RecipeItemLane1 := 'BLACK';
	ELSIF SorterControl.Par.LaneAllocationRecipe.Lane1ProductType = ptMETAL THEN
		RecipeItemLane1 := 'METAL';
	END_IF
	IF SorterControl.Par.LaneAllocationRecipe.Lane2ProductType = ptRED THEN
		RecipeItemLane2 := 'RED';
	ELSIF SorterControl.Par.LaneAllocationRecipe.Lane2ProductType = ptBLACK THEN
		RecipeItemLane2 := 'BLACK';
	ELSIF SorterControl.Par.LaneAllocationRecipe.Lane2ProductType = ptMETAL THEN
		RecipeItemLane2 := 'METAL';
	END_IF
	IF SorterControl.Par.LaneAllocationRecipe.Lane3ProductType = ptRED THEN
		RecipeItemLane3 := 'RED';
	ELSIF SorterControl.Par.LaneAllocationRecipe.Lane3ProductType = ptBLACK THEN
		RecipeItemLane3 := 'BLACK';
	ELSIF SorterControl.Par.LaneAllocationRecipe.Lane3ProductType = ptMETAL THEN
		RecipeItemLane3 := 'METAL';
	END_IF

	AutomaticMode;
	HomingMode;
	ManualMode;

	gReset := ResetMode;

	TimeStruct;

	TIME_TO_TIMEStructure(AutomaticGeneralInfo.AutomaticModeTime, ADR(TimeStruct));

END_PROGRAM

PROGRAM _EXIT

END_PROGRAM
```

#### Types.typ - Local data types
```iecst
(*local enum types*)

TYPE
	OpModeEnum :
		( (*Enumerated type for state machine*)
		omMANUAL, (*Manual mode*)
		omAUTOMATIC, (*Automatic mode*)
		omHOMING (*Homing mode*)
		);
END_TYPE
```

#### Variables.var - Local variables
```iecst
(*local variables*)
VAR
	AutomaticActive : BOOL; (*Tracker to see if Automatic is active*)
	AutomaticMode : BOOL := FALSE; (*Automatic mode variable*)
	ManualMode : BOOL := FALSE; (*Manual mode variable*)
	HomingMode : BOOL := FALSE; (*Homing mode variable*)
	ActiveMode : STRING[100]; (*Active mode of the machine*)
	StartMode : BOOL; (*Start command*)
	StopMode : BOOL; (*Stop command*)
	ResetMode : BOOL; (*Reset command*)
	ErrorMessageMainPage : STRING[255]; (*Error message on Main page*)
	OpModeState : OpModeEnum := 0; (*Operational mode enumerator state machine*)
	ErrorMessageManualPage : STRING[255]; (*Error message variable for Manual page*)
	ProductRed : BOOL; (*Product is red*)
	ProductBlack : BOOL; (*Product is black*)
	ProductMetal : BOOL; (*Product is metal*)
	RequiredSwitch : STRING[255] := 'No product identified'; (*Switch required based on lane selection*)
	AutoIdentifiedProduct : BOOL; (*Bit for when product is identified*)
	RecipeItemLane1 : STRING[255]; (*String rep of color of lane*)
	ManualEnable : BOOL; (*Boolean to enable manual mode*)
	RecipeItemLane2 : STRING[255]; (*String rep of color of lane*)
	RecipeItemLane3 : STRING[255]; (*String rep of color of lane*)
	TimeStruct : TIMEStructure; (*Time structure*)
	SortingStationStatus : STRING[255] := 'Sorting station starting up, please home machine before starting Automatic Mode'; (*Sorting station status message*)
	SortingHomed : BOOL;
END_VAR
```

### Package Logical/Infrastructure/Comms - OPCUA communication

### CommsIF.typ - Comms interface types
```iecst
(*global interface variables for comms*)

TYPE
	OpcUaWriteType : 	STRUCT  (*Variables that are written to the Distribution Station*)
		ConveyorVelocity : REAL;
	END_STRUCT;
	OpcUaReadType : 	STRUCT  (*Variables that are read from the Distribution Station*)
		ProductArriving : BOOL; (*Product is arriving at the Sorting Station*)
		DistributionReady : BOOL; (*Distribution station is ready*)
		DistributionHomed : BOOL; (*Station is homed*)
		HomingConfirm : BOOL; (*Homing done confirmation button pressed*)
		AutomaticActive : BOOL; (*TRUE if automatic is controlled from Distribution station*)
	END_STRUCT;
	OpcUaControlType : 	STRUCT
		Write : OpcUaWriteType; (*Write variables*)
		Read : OpcUaReadType; (*Read variables*)
		ServerConnectionError : BOOL; (*Server communcication error*)
	END_STRUCT;
END_TYPE
```

### CommsIF.var - Comms interface vars
```iecst
(*global interface variables*)
VAR
	OpcUaControl : OpcUaControlType; (*Control structure for OPCUA*)
END_VAR
```

### Program Logical/Infrastructure/Comms/Comms (IEC) - Communications task

#### Main.st - Init, cyclic, exit code
```iecst
(*********************************************************************************
 * Copyright:   B&R Industrial Automation GmbH
 * Author:      lauryr
 * Created:     May 19, 2025/5:55 PM
 * Description: Basic program to interact with the Distribution Station via OPCUA
 *********************************************************************************)

PROGRAM _INIT
	(* Insert code here *)

END_PROGRAM

PROGRAM _CYCLIC
	(* Insert code here *)

	OpcUaControl;

	IF NOT OpcUaControl.Read.DistributionReady THEN
		gStop := TRUE;
	ELSE
		IF gStop THEN
			gStop := FALSE;
		END_IF
END_IF

END_PROGRAM

PROGRAM _EXIT
	(* Insert code here *)

END_PROGRAM
```

### Package Logical/Documentation - Package containing project documentation

- Visualisation Logical/mappView (not shown)
